   REGION External Keys /LED
       // Start Cycle
       #sStartCycle(iKeyHWStatus := "DI_PB_StartCycle",
                    oLedHWStatus => "DQ_StartCycleGreenLED");

       // Alarm Reset
       #sAlarmReset(iKeyHWStatus := "DI_PB_ResetAlarm",
                    oLedHWStatus => "DQ_AlarmBlueLED");

       // Power OFF
       #sPowerOFF(iKeyHWStatus := "DI_PB_PowerOFF",
                  oLedHWStatus => #tNoLed);

       // Shutdown PC
       #sShutdownPC(iKeyHWStatus := "DI_PB_ShutdownPC",
                    oLedHWStatus => "DQ_ShutdownPCYellowLED");

       // Light Test
       #sLightTest(iKeyHWStatus := "DI_PB_LightTest",
                   oLedHWStatus => "DQ_LightTestWhiteLED");

       // Power ON
       #sPowerON(iKeyHWStatus := "DI_PB_PowerON",
                 oLedHWStatus => "DQ_PowerOnGreenLED");

       // Remote Open Shutter
       #sRemoteOpenShutter(iKeyHWStatus := "DI_PB_RemoteOpenShutter",
                           oLedHWStatus => "DQ_RemoteOpenShutterWhiteLED");
   END_REGION

   REGION Axis Keys (Right Panel)
       #sAx10_LaserArea(iKeyHWStatus := "MCP1_In".axis10,
                        oLedHWStatus => "MCP1_Out".LEDaxis10);

       #sAx11_ChannelSelection(iKeyHWStatus := "MCP1_In".axis11,
                               oLedHWStatus => "MCP1_Out".LEDaxis11);
   END_REGION
END_FUNCTION_BLOCK

FUNCTION_BLOCK "FB_McpKeysSignals"   // FB422, SCL
{ S7_Optimized_Access := 'TRUE' }
// stored: AutoNumber false, MemoryReserve 100, SetENOAutomatically false
   VAR_INPUT
      iKeyHWStatus { ExternalAccessible := 'False'; ExternalVisible := 'False'; ExternalWritable := 'False'} : Bool;   // PLC Digital Input Hardware status
   END_VAR
   VAR_OUTPUT
      oLedHWStatus : Bool;
   END_VAR
   VAR
      sKeySWStatus : Bool;
      sKeySWToggleStatus : Bool;
      sKeyDisable : Bool;
      sKeySWPositiveFront : Bool;
      sKeySWNegativeFront : Bool;
      sKeySWTogglePositiveFront : Bool;
      sKeySWToggleNegativeFront : Bool;
      sLedSWStatus : Bool;
      sRT_KeySWPositiveFront { S7_SetPoint := 'True'} : R_TRIG;
      sFT_KeySWNegativeFront { S7_SetPoint := 'True'} : F_TRIG;
      sRT_KeySWTogglePositiveFront { S7_SetPoint := 'True'} : R_TRIG;
      sFT_KeySWToggleNegativeFront { S7_SetPoint := 'True'} : F_TRIG;
   END_VAR
BEGIN
   REGION Description header 
       //==================================================================================
       // POSALUX Swiss SA / (C) Copyright 2025
       //----------------------------------------------------------------------------------
       // Title: Management of inputs and outputs for MCP and external buttons 
       // Comment/Function: 
       //
       // Author: Fabien Waldt
       // Engineering: TIA Portal v19
       //----------------------------------------------------------------------------------
       // Change log table:
       // Version  | Date     | Expert in charge | Changes applied
       // ---------|----------|------------------|------------------------------------
       // 00.00.01 | 20250911 | WFA              | First released version
       // 00.00.02 | 20260218 | WFA              | Remove reset toggle when disable
       // ==================================================================================
   END_REGION

   REGION Inputs keys
           // Management of inputs for each customerkey MCP button 
           // Management of the software input
            IF NOT #sKeyDisable THEN
                #sKeySWStatus := #iKeyHWStatus;
            END_IF;

           // Rising/falling edge detection when pressing the button
           #sRT_KeySWPositiveFront(CLK := #sKeySWStatus,
                                  Q => #sKeySWPositiveFront);

           #sFT_KeySWNegativeFront(CLK := #sKeySWStatus,
                                  Q => #sKeySWNegativeFront);

           // Toggle state update
           IF #sKeySWPositiveFront  THEN
               #sKeySWToggleStatus := NOT #sKeySWToggleStatus;
           END_IF;

           // Rising/falling edge detection of the toggle state
           #sRT_KeySWTogglePositiveFront(CLK := #sKeySWToggleStatus,
                                        Q => #sKeySWTogglePositiveFront);

           #sFT_KeySWToggleNegativeFront(CLK := #sKeySWToggleStatus,
                                        Q => #sKeySWToggleNegativeFront);
   END_REGION

   REGION Outputs LED   
       #oLedHWStatus := #sLedSWStatus;
   END_REGION
END_FUNCTION_BLOCK

FUNCTION_BLOCK "FB_LaserAirProcess"   // FB432, SCL
{ S7_Optimized_Access := 'TRUE' }
// stored: AutoNumber false, MemoryReserve 100, SetENOAutomatically false
   VAR
      sTimeDelay : Time;
      sTimerGas : TON_TIME;
      sGasAssistOn : Bool;
      sLaser_Air_Process_Ctrl { S7_SetPoint := 'True'} : "FB_AnalogInputThreshold";
      sNozzle_Over_Pressure { S7_SetPoint := 'True'} : "FB_AnalogInputThreshold";
      sGasAssistDelay { ExternalAccessible := 'False'; ExternalVisible := 'False'; ExternalWritable := 'False'} : Bool;
      sGasAssistStartCh1 : Bool;
      sGasAssistStartCh2 : Bool;
      sGasAssistByKey : Bool;
      sGasReadValue : Bool;
      sRT_sGasAssistStartCh1 : R_TRIG;
      sRT_sGasAssistStartCh2 { S7_SetPoint := 'True'} : R_TRIG;
      sFT_sGasAssistStartCh1 { S7_SetPoint := 'True'} : F_TRIG;
      sFT_sGasAssistStartCh2 { S7_SetPoint := 'True'} : F_TRIG;
      sGasAssistSetPointJog { S7_SetPoint := 'True'} : Real;
      sGasAssistOffTimer : TOF_TIME;
   END_VAR
   VAR_TEMP
      tReadError : Bool;
      tErrorCode : Int;
   END_VAR
   VAR CONSTANT
      GAS_ASSIST_TIME : Time := T#5m;
   END_VAR
BEGIN
   REGION Description header 
       //==================================================================================
       // POSALUX Swiss SA / (C) Copyright 2024
       //----------------------------------------------------------------------------------
       // Title: Laser AirProcess
       // Comment/Function: 
       //
       // Author: Gowsigan SRITHARAN
       // Engineering: TIA Portal v17
       //----------------------------------------------------------------------------------
       // Change log table:
       // Version  | Date     | Expert in charge | Changes applied
       // ---------|----------|------------------|------------------------------------
       // 00.00.01 | 20241205 | GSR              | First released version
       // 00.00.02 | 20250314 | WFA              | Management modifications in Jog Mode
       // ==================================================================================
   END_REGION

   REGION Gas Assist ON
       "DB_DigitalOutputs".sGasAssistOn.sSWStatus := "DB_PowerOn".sMachineReadySoft;
   END_REGION

   REGION Disable Gas Assist Key[2]
       "DB_McpKeyboardSignals".sK2_GasAssist.sKeyDisable :=
       NOT "LBP_ModeGroup".E_JOG
       OR "LBP_Chan1".E_ProgRunning
       OR "LBP_Chan1".E_ProgStop
       OR "LBP_Chan1".E_ProgWait
       OR "DB_GestionWorkingModes".sMCP_KxxKeysDisable;

       "DB_HmiKeyboardSignals".sK2_GasAssist.sKeyDisable :=
       NOT "LBP_ModeGroup".E_JOG
       OR "LBP_Chan1".E_ProgRunning
       OR "LBP_Chan1".E_ProgStop
       OR "LBP_Chan1".E_ProgWait;
   END_REGION

   REGION Gas Assist
       IF "LBP_Chan1".MDyn[90] THEN                                // M90 : Start Gas Assist
           #sGasAssistStartCh1 := TRUE;
       ELSIF "LBP_Chan1".MDyn[91] OR "LBP_Chan1".A_Reset THEN      // M91 : Stop Gas Assist
           #sGasAssistStartCh1 := FALSE;
       END_IF;
   END_REGION

   REGION Gas Assist by Key
       IF "DB_McpKeyboardSignals".sK2_GasAssist.sKeySWTogglePositiveFront
           OR "DB_HmiKeyboardSignals".sK2_GasAssist.sKeySWTogglePositiveFront THEN
           #sGasAssistByKey := TRUE;
       ELSIF "DB_McpKeyboardSignals".sK2_GasAssist.sKeySWToggleNegativeFront
           OR "DB_HmiKeyboardSignals".sK2_GasAssist.sKeySWToggleNegativeFront THEN
           #sGasAssistByKey := FALSE;
       END_IF;
   END_REGION

   REGION Gas Read Value
       #sRT_sGasAssistStartCh1(CLK := #sGasAssistStartCh1);
       #sFT_sGasAssistStartCh1(CLK := #sGasAssistStartCh1);

       IF #sRT_sGasAssistStartCh1.Q
           OR #sFT_sGasAssistStartCh1.Q THEN
               #sGasReadValue := TRUE;
       END_IF;
   END_REGION

   REGION Nitrogen Gas LED[2]
       "DB_McpKeyboardSignals".sK2_GasAssist.sLedSWStatus :=
       #sGasAssistStartCh1
       OR #sGasAssistByKey;

       "DB_HmiKeyboardSignals".sK2_GasAssist.sLedSWStatus :=
       #sGasAssistStartCh1
       OR #sGasAssistByKey;
   END_REGION

   REGION Laser Air Pressure Process Set Point
       "DB_DigitalOutputs".sLaserAirPressureProcess.sSWStatus :=
       #sGasAssistStartCh1
       OR #sGasAssistByKey;
   END_REGION

   REGION Gas Assist Set point
       "LBP_TransferSelData"(Enable := #sGasReadValue,
                             Funct := 16#03,
                             IVAR1 := 972,
                             IVAR2 := -1,
                             Error => #tReadError,
                             ErrCode => #tErrorCode,
                             S7Var := "DB_HMISetting".GasAssistSetPoint);

       // Gas Assist Set Point if Jog mode
       IF NOT "LBP_ModeGroup".E_JOG AND "DB_HMISetting".GasAssistSetPoint <> 0 AND #sGasReadValue THEN
           #sGasAssistSetPointJog := "DB_HMISetting".GasAssistSetPoint;
       ELSE
           #sGasAssistSetPointJog := "DB_Parameters".GazPressureManual;
        END_IF;   

       // Transfer Gas Assist Set Point
        IF #sGasReadValue THEN
           IF "LBP_ModeGroup".E_JOG THEN
               "DB_AnalogInputDataHMI".Laser_Air_Pressure_Process.TargetValue := #sGasAssistSetPointJog;
               "DB_AnalogInputDataHMI".Nozzle_Overpressure.TargetValue := #sGasAssistSetPointJog;
           ELSE
               "DB_AnalogInputDataHMI".Laser_Air_Pressure_Process.TargetValue := "DB_HMISetting".GasAssistSetPoint;
               "DB_AnalogInputDataHMI".Nozzle_Overpressure.TargetValue := "DB_HMISetting".GasAssistSetPoint;
           END_IF;
       END_IF;

       // Reset Gas Assist Value by push Reset Button or after 5min no process
       #sGasAssistOffTimer(IN := ("LBP_Chan1".E_ProgRunning AND "LBP_Chan1".E_ProgRunning)
                           OR ("LBP_ModeGroup".E_JOG AND "DB_McpKeyboardSignals".sK2_GasAssist.sKeySWToggleStatus)
                           OR ("LBP_ModeGroup".E_JOG AND "DB_HmiKeyboardSignals".sK2_GasAssist.sKeySWToggleStatus),
                           PT := #GAS_ASSIST_TIME);

       // IF "MCP1_In".reset OR NOT #sGasAssistOffTimer.Q THEN
           IF "MCP1_In".reset THEN // WFA A REVOIR
           "DB_HMISetting".GasAssistSetPoint := 0.0;
           "DB_AnalogInputDataHMI".Laser_Air_Pressure_Process.TargetValue := 0.0;
           "DB_AnalogInputDataHMI".Nozzle_Overpressure.TargetValue := 0.0;
       END_IF;

       // Gas assist transfer to analog output
       IF NOT "LBP_ModeGroup".E_JOG THEN
           "DB_AnalogOutputs".sNozzleOverpressureSetPoint.sSWRealValue := "DB_HMISetting".GasAssistSetPoint;
       ELSE
           "DB_AnalogOutputs".sNozzleOverpressureSetPoint.sSWRealValue := #sGasAssistSetPointJog;
       END_IF;
   END_REGION

   REGION Laser Air process control
       #sLaser_Air_Process_Ctrl(iActualValue := "DB_AnalogInputs".sLaserAirPressureProcess.sSWRealValue,
                                iStartDelay := "DB_DigitalOutputs".sLaserAirPressureProcess.sSWStatus,
                                ioAlarmMin := "LBP_AlarmMsgs".UserA[06].A70UUxx[50],
                                ioWarningMin := "LBP_AlarmMsgs".UserA[07].A70UUxx[50],
                                ioWarningMax := "LBP_AlarmMsgs".UserA[07].A70UUxx[51],
                                ioAlarmMax := "LBP_AlarmMsgs".UserA[06].A70UUxx[51],
                                oDataAction => "DB_AnalogInputAction".Laser_Air_Pressure_Process,
                                iDataPLC := "DB_AnalogInputDataPLC".Laser_Air_Pressure_Process,
                                iDataHMI := "DB_AnalogInputDataHMI".Laser_Air_Pressure_Process);
     END_REGION

     REGION Regulation gas assist control
         #sNozzle_Over_Pressure(iActualValue := "DB_AnalogInputs".sNozzleOverpressure.sSWRealValue,
                                iStartDelay := "DB_DigitalOutputs".sLaserAirPressureProcess.sSWStatus,
                                ioAlarmMin := "LBP_AlarmMsgs".UserA[06].A70UUxx[60],
                                ioWarningMin := "LBP_AlarmMsgs".UserA[07].A70UUxx[60],
                                ioWarningMax := "LBP_AlarmMsgs".UserA[07].A70UUxx[61],
                                ioAlarmMax := "LBP_AlarmMsgs".UserA[06].A70UUxx[61],
                                oDataAction => "DB_AnalogInputAction".Nozzle_Overpressure,
                                iDataPLC := "DB_AnalogInputDataPLC".Nozzle_Overpressure,
                                iDataHMI := "DB_AnalogInputDataHMI".Nozzle_Overpressure);
     END_REGION
END_FUNCTION_BLOCK

FUNCTION_BLOCK "FB_AnalogInputThreshold"   // FB221, SCL
{ S7_Optimized_Access := 'TRUE' }
// stored: AutoNumber false, MemoryReserve 100, SetENOAutomatically false
   VAR_INPUT
      iActualValue : Real;
      iStartDelay : Bool;
      iDataPLC { ExternalAccessible := 'False'; ExternalVisible := 'False'; ExternalWritable := 'False'} : "AnalogInDataPLC_DT";
      iDataHMI { ExternalAccessible := 'False'; ExternalVisible := 'False'; ExternalWritable := 'False'} : "AnalogInDataHMI_DT";
   END_VAR
   VAR_OUTPUT
      oDataAction { ExternalAccessible := 'False'; ExternalVisible := 'False'; ExternalWritable := 'False'} : "AnalogInAction_DT";
   END_VAR
   VAR_IN_OUT
      ioAlarmMin : Bool;
      ioWarningMin : Bool;
      ioWarningMax : Bool;
      ioAlarmMax : Bool;
   END_VAR
   VAR
      sStartTimer : TON_TIME;
      sTONAlarmMin : TON_TIME;
      sTONWarningMin : TON_TIME;
      sTONWarningMax : TON_TIME;
      sTONAlarmMax : TON_TIME;
      sMemoAlarmMin { S7_SetPoint := 'True'} : Bool;
      sMemoWarningMin { S7_SetPoint := 'True'} : Bool;
      sMemoWarningMax { S7_SetPoint := 'True'} : Bool;
      sMemoAlarmMax { S7_SetPoint := 'True'} : Bool;
   END_VAR
BEGIN
   REGION Description header 
       //==================================================================================
       // POSALUX Swiss SA / (C) Copyright 2024
       //----------------------------------------------------------------------------------
       // Title: Analog input management 
       // Comment/Function: This function manages alarms and warnings based on a  
       //                   current value compared to predefined target. After an
       //                   initial delay, it activates specific alarms OR warnings if the
       //                   value exceeds thresholds, and can also trigger machine
       //                   shutdown or signal a defective part according TO conditions
       //                   configured on the HMI.
       // Author: Gowsigan SRITHARAN
       // Engineering: TIA Portal v17
       //----------------------------------------------------------------------------------
       // Change log table:
       // Version  | Date     | Expert in charge | Changes applied
       // ---------|----------|------------------|------------------------------------
       // 00.00.01 | 20241121 | GSR              | First released version
       // 00.00.02 | 20250911 | WFA              | Work with target
       // ==================================================================================
   END_REGION

   REGION Start Timer
       #sStartTimer(IN := #iStartDelay,
                    PT := #iDataHMI.StartTime);
       #sTONAlarmMin(IN := #sMemoAlarmMin,
                     PT := #iDataPLC.DelayAlarmMin);
       #sTONWarningMin(IN := #sMemoWarningMin,
                       PT := #iDataPLC.DelayWarningMin);
       #sTONAlarmMax(IN := #sMemoAlarmMax,
                     PT := #iDataPLC.DelayAlarmMax);
       #sTONWarningMax(IN := #sMemoWarningMax,
                       PT := #iDataPLC.DelayWarningMax);
   END_REGION

   REGION Detect alarm/warning
       IF #sStartTimer.Q THEN
           #sMemoWarningMin := #iDataHMI.TargetValue + #iDataHMI.ThresholdWarningMin >= #iActualValue AND #iDataPLC.EnableWarningMin AND NOT #sMemoAlarmMin;

           #sMemoWarningMax := #iDataHMI.TargetValue + #iDataHMI.ThresholdWarningMax <= #iActualValue AND #iDataPLC.EnableWarningMax AND NOT #sMemoAlarmMax;

           #sMemoAlarmMin := #iDataHMI.TargetValue + #iDataHMI.ThresholdAlarmMin >= #iActualValue AND #iDataPLC.EnableAlarmMin;

           #sMemoAlarmMax := #iDataHMI.TargetValue + #iDataHMI.ThresholdAlarmMax <= #iActualValue AND #iDataPLC.EnableAlarmMax;
       ELSE
           #sMemoWarningMin := FALSE;
           #sMemoWarningMax := FALSE;
           #sMemoAlarmMin   := FALSE;
           #sMemoAlarmMax   := FALSE;
       END_IF;

   END_REGION

   REGION Set alarm/warning
       // Alarme Min
       IF #sTONAlarmMin.Q THEN
           #ioAlarmMin := TRUE;
           #ioWarningMin := FALSE;
           #oDataAction.BadPartOnFixture := #iDataPLC.BadPartOnFixture; // Set bad part if alarm
           #oDataAction.ID_Measure := #iDataHMI.ID_Measure;
       ELSE
           #oDataAction.BadPartOnFixture := FALSE;
           #oDataAction.ID_Measure := 0;
       END_IF;

       // Warning Min
       IF #sTONWarningMin.Q THEN
           #ioWarningMin := TRUE;
       END_IF;

       // Alarm Max
       IF #sTONAlarmMax.Q THEN
           #ioAlarmMax := TRUE;
           #ioWarningMax := FALSE;
           #oDataAction.BadPartOnFixture := #iDataPLC.BadPartOnFixture; // Set bad part if alarm
           #oDataAction.ID_Measure := #iDataHMI.ID_Measure;
       ELSE
           #oDataAction.BadPartOnFixture := FALSE;
           #oDataAction.ID_Measure := 0;
       END_IF;

       // Warning Max
       IF #sTONWarningMax.Q THEN
           #ioWarningMax := TRUE;
       END_IF;
   END_REGION
END_FUNCTION_BLOCK

FUNCTION_BLOCK "FB_LaserOperation"   // FB431, SCL
{ S7_Optimized_Access := 'TRUE' }
// stored: AutoNumber false, MemoryReserve 100, SetENOAutomatically false
   VAR
      sLaserTimeCh1 : "FB_TimeCounter";
      sLaserCycleTimeCh1 { S7_SetPoint := 'True'} : Int;
   END_VAR
BEGIN
   REGION Description header 
       //==================================================================================
       // POSALUX Swiss SA / (C) Copyright 2024
       //----------------------------------------------------------------------------------
       // Title: Laser AirProcess
       // Comment/Function: 
       //
       // Author: Gowsigan SRITHARAN
       // Engineering: TIA Portal v17
       //----------------------------------------------------------------------------------
       // Change log table:
       // Version  | Date     | Expert in charge | Changes applied
       // ---------|----------|------------------|------------------------------------
       // 00.00.01 | 20241205 | GSR              | First released version
       // ==================================================================================
   END_REGION

   REGION Head Laser Circuit breaker
       IF NOT "DB_DigitalInputs".sHeadLaserBreaker.sSWStatus THEN
           "LBP_AlarmMsgs".UserA[0].A70UUxx[2] := TRUE;
       END_IF;
   END_REGION

   REGION Head_Laser start and stop
       "DB_DigitalOutputs".sHeadLaserStart.sSWStatus := "DB_PowerOn".sMachineReadySoft;
       "DB_DigitalOutputs".sHeadLaserStop.sSWStatus  := "DB_PowerOn".sMachineReadySoft;
   END_REGION

   REGION LED laser button 
       IF ("DB_DataFromSafety".ShutterOpened
           AND NOT "DB_DataFromSafety".ShutterClosed)
           OR "DB_McpKeyboardSignals".sLightTest.sKeySWStatus THEN  // Test Lamp
           "DB_McpKeyboardSignals".sRemoteOpenShutter.sLedSWStatus := TRUE;
       ELSIF "DB_DataFromSafety".ShutterClosed AND NOT "DB_DataFromSafety".ShutterOpened THEN
           IF "DB_DataFromSafety".ShutterReadyToOpen THEN
               // Ready to open -> slow blinking
               "DB_McpKeyboardSignals".sRemoteOpenShutter.sLedSWStatus := "Clock_0.5Hz";
           ELSIF "DB_DataFromSafety".OpenShutter THEN
               // Ready to open -> quick blinking
               "DB_McpKeyboardSignals".sRemoteOpenShutter.sLedSWStatus := "Clock_2Hz";
           ELSE
               // Close -> off
               "DB_McpKeyboardSignals".sRemoteOpenShutter.sLedSWStatus := FALSE;
           END_IF;
       ELSE
           // Close -> off
           "DB_McpKeyboardSignals".sRemoteOpenShutter.sLedSWStatus := FALSE;
       END_IF;
   END_REGION

   REGION Laser Key ON / Shutter closed
       "DB_HMIStatus".KeyLaserOn := "DB_DataFromSafety".iKeyLaserOn;
       "DB_HMIStatus".Shutter_laser_closed := "DB_DigitalInputs".sShutterClosed.sSWStatus OR NOT "DB_DataFromSafety".iKeyLaserOn;
   END_REGION


   REGION Laser Cycle Time
       #sLaserTimeCh1(iStart := "LBP_Chan1".MDyn[71],                        // M71 : Start calculation laser time 
                      iReset := "LBP_Chan1".MDyn[68] OR "MCP1_In".reset);    // M68 : Reset calculation laser time 
       #sLaserCycleTimeCh1 := #sLaserTimeCh1.ioMinutesCumul;
   END_REGION
END_FUNCTION_BLOCK

FUNCTION_BLOCK "FB_TimeCounter"   // FB53, SCL
{ S7_Optimized_Access := 'TRUE' }
// stored: MemoryReserve 100, SetENOAutomatically false
   VAR_INPUT
      iStart : Bool;
      iReset : Bool;
   END_VAR
   VAR_IN_OUT
      ioHours : Int;
      ioMinutes : Int;
      ioSeconds : Int;
      ioHoursCumul : Int;
      ioMinutesCumul : Int;
      ioSecondsCumul : DInt;
   END_VAR
   VAR
      sRT_Second { ExternalAccessible := 'False'; ExternalVisible := 'False'; ExternalWritable := 'False'} : R_TRIG;
   END_VAR
BEGIN
   REGION Description header 
       //==================================================================================
       // POSALUX Swiss SA / (C) Copyright 2025
       //----------------------------------------------------------------------------------
       // Title: Timer Counter
       // Comment/Function: This function allows:
       //                      - Counting Hours - Minutes - Seconds 
       //                      - Pulse each Hour - Minute - Second
       //
       // Author: Fabien Waldt
       // Engineering: TIA Portal v17
       //----------------------------------------------------------------------------------
       // Change log table:
       // Version  | Date     | Expert in charge | Changes applied
       // ---------|----------|------------------|------------------------------------
       // 00.00.01 | 20250314 | WFA              | First released version
       // ==================================================================================
   END_REGION

   //"Seconds" rising edge
   #sRT_Second(CLK := "Clock_1Hz");

   REGION Time counters reset
       IF #iReset THEN
           #ioHours := 0;
           #ioMinutes := 0;
           #ioSeconds := 0;
           #ioHoursCumul := 0;
           #ioMinutesCumul := 0;
           #ioSecondsCumul := 0;
       END_IF;
   END_REGION

   REGION Time counters
   IF #iStart AND #sRT_Second.Q THEN
       #ioSeconds := #ioSeconds + 1;
       #ioSecondsCumul := #ioSecondsCumul + 1;
       IF #ioSeconds >= 60 THEN
           #ioMinutes := #ioMinutes + 1;
           #ioSeconds := 0;
           #ioMinutesCumul := #ioMinutesCumul + 1;
           IF #ioMinutes >= 60 THEN
               #ioHours := #ioHours + 1;
               #ioMinutes := 0;
               #ioHoursCumul := #ioHoursCumul + 1;
           END_IF;
       END_IF;
   END_IF;
   END_REGION
END_FUNCTION_BLOCK

FUNCTION_BLOCK "FB_LaserMeasureZoneSwitch"   // FB417, SCL
{ S7_Optimized_Access := 'TRUE' }
// stored: AutoNumber false, MemoryReserve 100, SetENOAutomatically false
   VAR RETAIN
      sMeasure1 : Bool;   // Limit sw Measure 1 / Axes are on Area Measure station 1
      sMeasure2 : Bool;   // Limit sw Measure 2 / Axes are on Area Measure station 2
      sLaser1 : Bool;   // Condition Laser 1 / Gate for going to area laser Station 1
      sLaser2 : Bool;   // Condition Laser 2 / Gate for going to area laser Station 2
      sLaserArea1Req : Bool;   // Laser area 1 request / Ask for going to laser Area Station 1
      sLaserArea2Req : Bool;   // Laser area 2 request / Ask for going to laser Area Station 2
      sCuttingArea1Req : Bool;   // Cutting 1 request / Axe X1 enter to laser Area
      sCuttingArea2Req : Bool;   // Cutting 2 request / Axe X2 enter to laser Area
      sCutBusy : Bool;   // ???
      sCut1 : Bool;   // Axe X1 traverse the gate (X1SoftLimMin1)
      sCut2 : Bool;   // Axe X2 traverse the gate (X1SoftLimMin1)
      sX1Pos : Real;
      sX2Pos : Real;
   END_VAR
   VAR
      sRT_GateCut1 : R_TRIG;
      sRT_GateCut2 : R_TRIG;
   END_VAR
   VAR RETAIN
      sCondDegageAxe : Bool;
      sRefAxisActive : Bool;
   END_VAR
BEGIN
   REGION Description header 
       //==================================================================================
       // POSALUX Swiss SA / (C) Copyright 2025
       //----------------------------------------------------------------------------------
       // Title: FB_ManageLaserOrMeasureArea
       // Comment/Function: manages two zones (laser or measurement) on two statio
       // ns, if
       // present, based on the position of the axes and/or the state of a keyboard button.
       //It dynamically switches the software limits OF the axes (limit 1 OR 2) according
       //TO the active zone, allowing the machine’s safety AND behavior TO adapt TO each
       //operating mode.
       // Author: Fabien Waldt
       // Engineering: TIA Portal v17
       //----------------------------------------------------------------------------------
       // Change log table:
       // Version  | Date     | Expert in charge | Changes applied
       // ---------|----------|------------------|------------------------------------
       // 00.00.01 | 20250224 | FWA              | First released version
       // ==================================================================================
   END_REGION

   REGION Key [16] Disable + Toggle
       // Disable Key [16] - collision detection of the ZL axis with the X axis // WFA ??
       "DB_McpKeyboardSignals".sAx10_LaserArea.sKeyDisable := NOT "LBP_ModeGroup".E_JOG;
       //On channel change, update the MCP button to reflect the toggle status of the newly selected channel 
       // "DB_McpKeyboardSignals".Ax10_LaserArea.KeySWToggleStatus :=
       // (#LaserArea1Req AND "DB_DecodChannels".Chan1IsDisplayed);
   END_REGION

   REGION Laser Area 1 Request
       IF "LBP_Chan1".MDyn[60]     // M60: Axes Limit for Laser Area
           OR ("DB_McpKeyboardSignals".sAx10_LaserArea.sKeySWTogglePositiveFront  AND "DB_DecodChannels".sChan1IsDisplayed) THEN
           #sLaserArea1Req := TRUE;
           "LBP_AlarmMsgs".ChanA[1].RID_5C02xx[0] := TRUE;         // Msg: "510200 - Waiting gate laser - M60"
       END_IF;

       IF "LBP_Chan1".MDyn[61]     // M61: Axes Limit for Measure Area
           OR ("DB_McpKeyboardSignals".sAx10_LaserArea.sKeySWToggleNegativeFront AND "DB_DecodChannels".sChan1IsDisplayed) THEN
           #sLaserArea1Req := FALSE;
           "LBP_AlarmMsgs".ChanA[1].RID_5C02xx[1] := TRUE;    // Msg: "510201 - Waiting gate measure - M61"
       END_IF;


   END_REGION

   REGION Conditions to switch the limit of axis
       IF #sLaserArea1Req 
           AND ("DB_AxisPosition".sAxis03_ZM."$AA_IM" >= "DB_AxisPosition".sAxis03_ZM."$MA_POS_LIMIT_MINUS2")  // ZM upper as limit M2
           AND ("DB_AxisPosition".sAxis04_B."$AA_IM" >= "DB_AxisPosition".sAxis04_B."$MA_POS_LIMIT_MINUS2")    // B upper as limit M2
           AND ("DB_AxisPosition".sAxis07_V."$AA_IM" <= "DB_AxisPosition".sAxis07_V."$MA_POS_LIMIT_PLUS2")     // V below as limit P2
           AND ("DB_AxisPosition".sAxis02_Y."$AA_IM" <= "DB_AxisPosition".sAxis02_Y."$MA_POS_LIMIT_PLUS2")     // Y below as limit P2
           AND "DB_Powermeter".sPowermeterInHomePos THEN   // Powermeter retracted
               #sLaser1 := TRUE;    // Set Laser 1
               #sMeasure1 := FALSE;
      ELSIF NOT #sLaserArea1Req AND
          ("DB_AxisPosition".sAxis01_X."$AA_IM" <= "DB_AxisPosition".sAxis01_X."$MA_POS_LIMIT_PLUS") THEN   // X below as limit P1
               #sMeasure1 := TRUE;
               #sLaser1 := FALSE;
       ELSE
           #sMeasure1 := FALSE;
       END_IF;
   END_REGION

   REGION Switch of the limit of axis (laser --> limit 2 / Measure --> Limit 1)
       IF #sLaser1 THEN
           "LBP_Axis01_X".A_SWLimit2Plus := TRUE;
           "LBP_Axis02_Y".A_SWLimit2Plus := TRUE;
           "LBP_Axis03_ZM".A_SWLimit2Plus := TRUE;
           "LBP_Axis04_B".A_SWLimit2Plus := TRUE;
           "LBP_Axis07_V".A_SWLimit2Plus := TRUE;
       ELSIF #sMeasure1 THEN
           "LBP_Axis01_X".A_SWLimit2Plus := FALSE;
           "LBP_Axis02_Y".A_SWLimit2Plus := FALSE;
           "LBP_Axis03_ZM".A_SWLimit2Plus := FALSE;
           "LBP_Axis04_B".A_SWLimit2Plus := FALSE;
           "LBP_Axis07_V".A_SWLimit2Plus := FALSE;
       END_IF;
   END_REGION

   REGION Led of the MCP button

       "DB_McpKeyboardSignals".sAx10_LaserArea.sLedSWStatus :=
       ((#sLaserArea1Req AND #sLaser1)
       OR (#sLaserArea1Req AND NOT #sLaser1 AND "Clock_1Hz")
       OR (NOT #sLaserArea1Req AND NOT #sLaser1 AND "Clock_1Hz"))
       AND "DB_DecodChannels".sChan1IsDisplayed
       OR ((#sLaserArea2Req AND #sLaser2)
       OR (#sLaserArea2Req AND NOT #sLaser2 AND "Clock_1Hz")
       OR (NOT #sLaserArea2Req AND NOT #sLaser2 AND "Clock_1Hz"))
       AND "DB_DecodChannels".sChan2IsDisplayed;
   END_REGION

   REGION Read in disable
       // Read in disable: laser 1 : gate NOT ready
       IF NOT #sLaserArea1Req OR #sLaser1 OR "LBP_Chan1".A_Reset THEN
           "LBP_AlarmMsgs".ChanA[1].RID_5C02xx[0] := FALSE;
       END_IF;
       IF #sLaserArea1Req OR #sMeasure1 OR "LBP_Chan1".A_Reset THEN
           "LBP_AlarmMsgs".ChanA[1].RID_5C02xx[1] := FALSE;
       END_IF;
   END_REGION

   REGION Anticollision - A REVOIR LORS MISE EN ROUTE
       REGION Conditions de dégagement
           #sCondDegageAxe := "LBP_ModeGroup".E_JOG AND NOT "LBP_ModeGroup".E_REF;
       END_REGION

       REGION Machine en Ref Active
           #sRefAxisActive := "LBP_Chan1".A_Ref OR "LBP_Chan2".A_Ref;
       END_REGION

       REGION Anticollision entre X1/V1
           IF "LBP_Axis01_X".A_SWLimit2Minus// Ne sert plus a rien car 0<v<200 
               AND ("DB_AxisPosition".sAxis07_V."$AA_IM" >= 9999.9999) THEN
               "LBP_AlarmMsgs".Axis[01].FdStop[10] := TRUE;
               "LBP_AlarmMsgs".Axis[07].FdStop[10] := TRUE;
            //   "LBP_AlarmMsgs".UserA[2].A70UUxx[10] := TRUE;   // Msg: "702010 - ???"
           END_IF;
           //Pas compris pour eviter collision avec x1 et v1
           IF (#sCondDegageAxe AND "LBP_Axis07_V".E_TCMinus)
               OR NOT "DB_DataToSafety".FrontDoorLock
               OR #sRefAxisActive THEN
               "LBP_AlarmMsgs".Axis[01].FdStop[10] := FALSE;
               "LBP_AlarmMsgs".Axis[07].FdStop[10] := FALSE;
            //   "LBP_AlarmMsgs".UserA[2].A70UUxx[10] := FALSE;   // Msg: "702010 - ???"
           END_IF;
       END_REGION

       REGION Anticollision entre X1/ZM1
           IF "LBP_Axis01_X".A_SWLimit2Minus // Ne sert plus a rien car -22<ZM1<160 
               AND (9999.9999 <= "DB_AxisPosition".sAxis03_ZM."$AA_IM") THEN
               "LBP_AlarmMsgs".Axis[01].FdStop[10] := TRUE;
               "LBP_AlarmMsgs".Axis[03].FdStop[10] := TRUE;
            //   "LBP_AlarmMsgs".UserA[2].A70UUxx[11] := TRUE;   // Msg: "702011 - ???"
           END_IF;
           //Pas compris pour eviter collision avec x1 et v1
           IF (#sCondDegageAxe AND "LBP_Axis03_ZM".E_TCPlus)
               OR NOT "DB_DataToSafety".FrontDoorLock
               OR #sRefAxisActive THEN
               "LBP_AlarmMsgs".Axis[01].FdStop[10] := FALSE;
               "LBP_AlarmMsgs".Axis[03].FdStop[10] := FALSE;
          //   "LBP_AlarmMsgs".UserA[2].A70UUxx[11] := FALSE;   // Msg: "702011 - ???"
           END_IF;
       END_REGION
   END_REGION

   REGION Cutting
       // WFA VOIR SI CUTTING NECESSAIRE POUR MACHINE MONO
       REGION Cutting : M62 waiting laser cutting free
           IF "LBP_Chan1".MDyn[62] THEN    // M62: Axes Limit for Cutting Area
               #sCuttingArea1Req := TRUE;
               "LBP_AlarmMsgs".ChanA[1].RID_5C02xx[2] := TRUE;         // Msg: "510202 - Waiting laser"
               #sX1Pos := LREAL_TO_REAL("DB_AxisPosition".sAxis01_X."$AA_IM");
           END_IF;
       END_REGION

       REGION Set cutting busy by X pos : JOG, man, prog interrupt, prog err
           #sRT_GateCut1(CLK := "DB_AxisPosition".sAxis01_X."$AA_IM" < "DB_AxisPosition".sAxis01_X."$A1_M_FP_POS4_30600");
           IF #sRT_GateCut1.Q THEN
               #sCut1 := TRUE;
           END_IF;
       END_REGION

       REGION X collision avoid
           IF #sCut1 AND #sCut2 THEN
               "LBP_AlarmMsgs".Axis[1].FdStop[0] := TRUE;
               "LBP_AlarmMsgs".Axis[10].FdStop[0] := TRUE;
           END_IF;

           // X1 plus: R stop X1
           IF "LBP_Chan1".E_ChanReset
               OR "LBP_Axis01_X".E_TCPlus
               OR "LBP_Chan1".A_Reset
               OR ("LBP_ModeGroup".E_JOG AND "LBP_ModeGroup".E_REF) THEN
               "LBP_AlarmMsgs".Axis[1].FdStop[0] := FALSE;
           END_IF;
           //check programmed X destination position
           //if in cuting area without gate_cut:stop
       END_REGION

       REGION Open cutting laser gate
           IF #sCuttingArea1Req THEN
               #sCut1 := TRUE;
               // ZL Get -> chan 1
               "LBP_Axis09_ZL".A_NCASpStrobe := TRUE;
               "LBP_Axis09_ZL".A_NCASpChanB := FALSE;
               "LBP_Axis09_ZL".A_NCASpChanA := TRUE;
           END_IF;
       END_REGION
       REGION Reset Gate_Cut_1 and Gate_Cut_2
           IF #sX1Pos >= "DB_AxisPosition".sAxis01_X."$A1_M_FP_POS4_30600" THEN
               #sX1Pos := LREAL_TO_REAL("DB_AxisPosition".sAxis01_X."$A1_M_FP_POS4_30600");
           END_IF;

           IF #sX1Pos + 1.0 < "DB_AxisPosition".sAxis01_X."$AA_IM" OR
               "LBP_Chan1".MDyn[63] THEN
               #sCut1 := FALSE;
           END_IF;
       END_REGION

       REGION Release M62
           // IF #sCut1 AND
           //     "LBP_Axis09_ZL".E_NCASpChanA
           //     AND NOT "LBP_Axis09_ZL".E_NCASpChanB
           //     OR "LBP_Chan1".A_Reset THEN
           //     "LBP_Axis09_ZL".A_NCASpStrobe := FALSE;
           //     #sCuttingArea1Req := FALSE;
           IF "DB_OPC_Laser".Scanner.In.Ready THEN
               "LBP_AlarmMsgs".ChanA[1].RID_5C02xx[2] := FALSE;         // Msg: "510202 - Waiting laser"
           END_IF;
       END_REGION
   END_REGION
   //Copie de la FL0125, Pas sur que ca existe sur les FEMTO 5A mono ou twin
   //A voir egalement les colisions à partir du code de la FL0107

   // REGION NETWORK 34
   //     IF "LBP_Chan1".MDyn[62] THEN    // M62: Axes Limit for Cutting Area
   //         #CuttingArea1Req := TRUE;
   //         "LBP_AlarmMsgs".ChanA[1].RID_5C02xx[2] := TRUE;
   //         #X1_POS := LREAL_TO_REAL("DB_AxisPosition_ReadVar".sAxis01_X1."$AA_IM");
   //     END_IF;

   //     IF "LBP_Chan2".MDyn[62] THEN    // M62: Axes Limit for Cutting Area
   //         #CuttingArea2Req := TRUE;
   //         "LBP_AlarmMsgs".ChanA[2].RID_5C02xx[2] := TRUE;
   //         #X2_POS := LREAL_TO_REAL("DB_AxisPosition_ReadVar".sAxis10_X2."$AA_IM");
   //     END_IF;
   // END_REGION

   // REGION NETWORK 35
   //     // WFA A REVOIR
   //     #Gate_Cut_1 := FALSE;
   //     #Gate_Cut_2 := FALSE;
   // END_REGION

   // REGION NETWORK 36
   //     IF #Gate_Cut_1 AND #Gate_Cut_2 THEN
   //         "LBP_AlarmMsgs".Axis[1].FdStop[0] := TRUE;
   //         "LBP_AlarmMsgs".Axis[10].FdStop[0] := TRUE;
   //     END_IF;

   //     //x1 plus: R stop x1
   //     IF "LBP_Chan1".E_ChanReset
   //         OR "LBP_Axis01_X1".E_TCPlus
   //         OR "LBP_Chan1".A_Reset
   //         OR ("LBP_ModeGroup".E_JOG AND "LBP_ModeGroup".E_REF) THEN
   //         "LBP_AlarmMsgs".Axis[1].FdStop[0] := FALSE;
   //     END_IF;

   //     //x2 minus: R stop x2
   //     IF "LBP_Chan2".E_ChanReset
   //         OR "LBP_Axis10_X2".E_TCMinus
   //         OR "LBP_Chan2".A_Reset
   //         OR ("LBP_ModeGroup".E_JOG AND "LBP_ModeGroup".E_REF) THEN
   //         "LBP_AlarmMsgs".Axis[10].FdStop[0] := FALSE;
   //     END_IF;


   //     //check programmed X destination position
   //     //if in cuting area without gate_cut:stop
   // END_REGION

   // REGION NETWORK 37
   //     IF #CuttingArea1Req AND NOT #Gate_Cut_2 THEN
   //         #Gate_Cut_1 := TRUE;
   //         "LBP_Axis09_ZL".A_NCASpStrobe := TRUE;
   //         "LBP_Axis09_ZL".A_NCASpChanB := FALSE;
   //         "LBP_Axis09_ZL".A_NCASpChanA := TRUE;
   //     END_IF;

   //     IF #CuttingArea2Req AND NOT #Gate_Cut_2 THEN
   //         #Gate_Cut_2 := TRUE;
   //         "LBP_Axis09_ZL".A_NCASpStrobe := TRUE;
   //         "LBP_Axis09_ZL".A_NCASpChanB := TRUE;
   //         "LBP_Axis09_ZL".A_NCASpChanA := FALSE;
   //     END_IF;
   // END_REGION

   // REGION NETWORK 38
   //     // WFA A REVOIR
   //     IF #X1_POS + 1.0 < "DB_AxisPosition_ReadVar".sAxis01_X1."$AA_IM" OR
   //         "LBP_Chan1".MDyn[63] THEN
   //         #Gate_Cut_1 := FALSE;
   //     END_IF;

   //     IF #X2_POS + 1.0 < "DB_AxisPosition_ReadVar".sAxis10_X2."$AA_IM" OR
   //         "LBP_Chan2".MDyn[63] THEN
   //         #Gate_Cut_2 := FALSE;
   //     END_IF;
   // END_REGION


   // REGION NETWORK 39
   //     IF #Gate_Cut_1 AND
   //         "LBP_Axis09_ZL".E_NCASpChanA
   //         AND NOT "LBP_Axis09_ZL".E_NCASpChanB
   //         OR "LBP_Chan1".A_Reset THEN
   //         "LBP_Axis09_ZL".A_NCASpStrobe := FALSE;
   //         #CuttingArea1Req := FALSE;
   //         "LBP_AlarmMsgs".ChanA[1].RID_5C02xx[2] := FALSE;
   //     END_IF;

   //     IF #Gate_Cut_2 AND
   //         NOT "LBP_Axis09_ZL".E_NCASpChanA
   //         AND "LBP_Axis09_ZL".E_NCASpChanB
   //         OR "LBP_Chan2".A_Reset THEN
   //         "LBP_Axis09_ZL".A_NCASpStrobe := FALSE;
   //         #CuttingArea2Req := FALSE;
   //         "LBP_AlarmMsgs".ChanA[2].RID_5C02xx[2] := FALSE;
   //     END_IF;
   // END_REGION
END_FUNCTION_BLOCK

FUNCTION_BLOCK "FB_Powermeter"   // FB433, SCL
{ S7_Optimized_Access := 'TRUE' }
// stored: AutoNumber false, MemoryReserve 100, SetENOAutomatically false
   VAR
      sPowerMeterWorkPos : Bool;
      sPowerMeterHomePos : Bool;
      sPowerMeterToWorkMoveReq : Bool;
      sPowerMeterToHomeMoveReq : Bool;
      sPowerMeterJogMode : Bool;
      sPowermeterCylinder : "FB_CmdCylinder";
      sPowermeterInHomePos { S7_SetPoint := 'True'} : Bool;
      sPowermeterInMiddlePos : Bool;
      sPowermeterInWorkPos : Bool;
      sPowerMeterCylErrorCode : Int;
      sPowerMeterHomePosCtrlTimer : TON_TIME;
      sPowerMeterWorkPosCtrlTimer : TON_TIME;
      sMeasurePowerLaser { S7_SetPoint := 'True'} : Bool;
      sRTLaserMeasureON : R_TRIG;
      sLaserPowerValue { S7_SetPoint := 'True'} : Real;
      sWeightFactor : Real;
      sAlpha : Real;
      sDateAndTime : DTL;
      sActualMeasPower : Real;
      sTolMin : Real;
      sTolMax : Real;
      sResetMeasures : Bool;
      sPowerMeterSeq : "FB_PowerMeterSeq";
      RT_StartArchive { S7_SetPoint := 'True'} : R_TRIG;
      sArchivePmValues { S7_SetPoint := 'True'} : Array[0..4] of Real;
   END_VAR
   VAR_TEMP
      tAxis01_X1SafePos : Bool;
      tLaserMeasureON : Bool;
      tActualMeasure : Int;
      tRetVal : Int;
      tAverageValue : Real;
      tStandardDeviation : Real;
      tTempReal : Real;
      tIndex : Int;
   END_VAR
   VAR CONSTANT
      POWERMETER_HOME_POS_CTRL_TIME : Time := T#6s;
      POWERMETER_WORK_POS_CTRL_TIME : Time := T#6s;
   END_VAR
BEGIN
   REGION Description header 
       //==================================================================================
       // POSALUX Swiss SA / (C) Copyright 2025
       //----------------------------------------------------------------------------------
       // Title: Initialization of axis
       // Comment/Function: 
       // Author: Fabien WALDT
       // Engineering: TIA Portal v17
       //----------------------------------------------------------------------------------
       // Change log table:
       // Version  | Date     | Expert in charge | Changes applied
       // ---------|----------|------------------|-----------------------------------------
       // 00.00.01 | 20250501 | WFA              | First released version
       // =================================================================================
   END_REGION

   REGION Axis01_X on safe position
      // Check position Axis01_X to release the powermeter
       #tAxis01_X1SafePos := "DB_AxisPosition".sAxis01_X."$AA_IM" >= "DB_AxisPosition".sAxis01_X."$MA_POS_LIMIT_PLUS" - 10.0;
   END_REGION

   REGION Blocking Axis01_X
       // Blocking Axis01_X if Powermeter is in measuring position
       "LBP_Axis01_X".A_ASpDisable := NOT #sPowerMeterHomePos OR #sPowerMeterWorkPos; 
   END_REGION
   REGION PowerMeter Sequence
       // #sPowerMeterSeq(iStartSeqCond:=#sPowerMeterSeq.iStartSeqCond,
       //                 iJobReq:=#sPowerMeterSeq.iJobReq,
       //                 iPowerMeterHomePos:=#sPowerMeterSeq.iPowerMeterHomePos,
       //                 iPowerMeterWorkPos:=#sPowerMeterSeq.iPowerMeterWorkPos,
       //                 iNC_Stopped:=#sPowerMeterSeq.iNC_Stopped,
       //                 iPLC_DateAndTime:="DB_ReadDateAndTime".sDateAndTime,
       //                 iStepPause:=#sPowerMeterSeq.iStepPause,
       //                 rMinValue:=#sPowerMeterSeq.rMinValue,
       //                 rMaxValue:=#sPowerMeterSeq.rMaxValue,
       //                 iStopOption:=#sPowerMeterSeq.iStopOption,
       //                 rMeasureValue:=#sPowerMeterSeq.rMeasureValue,
       //                 iMeasureDone:=#sPowerMeterSeq.iMeasureDone,
       //                 oPowerMetertoHomeReq=>#sPowerMeterSeq.oPowerMetertoHomeReq,
       //                 oPowerMetertoWorkReq=>#sPowerMeterSeq.oPowerMetertoWorkReq,
       //                 oStopNC_Req=>#sPowerMeterSeq.oStopNC_Req,
       //                 oMsgBadMeasure=>#sPowerMeterSeq.oMsgBadMeasure,
       //                 oStartMeasure=>#sPowerMeterSeq.oStartMeasure,
       //                 oStartArchive=>#sPowerMeterSeq.oStartArchive,
       //                 oRID=>#sPowerMeterSeq.oRID);
   END_REGION

   REGION Powermeter Key / LED Management
       // Disable Powemeter Key[1] if not Jog Mode
       "DB_McpKeyboardSignals".sK1_Powermeter.sKeyDisable := NOT "LBP_ModeGroup".E_JOG OR NOT #tAxis01_X1SafePos OR "DB_GestionWorkingModes".sMCP_KxxKeysDisable;
       "DB_HmiKeyboardSignals".sK1_Powermeter.sKeyDisable := NOT "LBP_ModeGroup".E_JOG OR NOT #tAxis01_X1SafePos;

       // Set/Reset Toggle Powemeter Key[1]
       IF #sPowerMeterSeq.oPowerMetertoWorkReq THEN    // Powermeter to work position
           "DB_McpKeyboardSignals".sK1_Powermeter.sKeySWToggleStatus := TRUE;
           "DB_HmiKeyboardSignals".sK1_Powermeter.sKeySWToggleStatus := TRUE;
       END_IF;
       IF #sPowerMeterSeq.oPowerMetertoHomeReq OR     // Powermeter to home position
           "LBP_Chan1".A_Reset  THEN
           "DB_McpKeyboardSignals".sK1_Powermeter.sKeySWToggleStatus := FALSE;
           "DB_HmiKeyboardSignals".sK1_Powermeter.sKeySWToggleStatus := FALSE;
           END_IF;

       // Powemeter LED[1] Animation
           "DB_McpKeyboardSignals".sK1_Powermeter.sLedSWStatus :=
           ("DB_McpKeyboardSignals".sK1_Powermeter.sKeySWToggleStatus AND #tAxis01_X1SafePos)
           OR ("DB_McpKeyboardSignals".sK1_Powermeter.sKeySWToggleStatus AND "Clock_2Hz");

           "DB_HmiKeyboardSignals".sK1_Powermeter.sLedSWStatus :=
           ("DB_HmiKeyboardSignals".sK1_Powermeter.sKeySWToggleStatus AND #tAxis01_X1SafePos)
           OR ("DB_HmiKeyboardSignals".sK1_Powermeter.sKeySWToggleStatus AND "Clock_2Hz");
   END_REGION

   REGION Powermeter in work position move request
       #sPowerMeterToWorkMoveReq :=
       ("DB_McpKeyboardSignals".sK1_Powermeter.sKeySWToggleStatus AND NOT "MCP1_In".incVar)
       OR ("DB_HmiKeyboardSignals".sK1_Powermeter.sKeySWToggleStatus AND NOT "MCP1_In".incVar)
       AND #tAxis01_X1SafePos;
   END_REGION

   REGION Powermeter in home position move request
       #sPowerMeterToHomeMoveReq :=
       (NOT "DB_McpKeyboardSignals".sK1_Powermeter.sKeySWToggleStatus AND
        NOT "DB_HmiKeyboardSignals".sK1_Powermeter.sKeySWToggleStatus);
   END_REGION

   REGION Powermeter in JOG Mode
       #sPowerMeterJogMode := "LBP_ModeGroup".E_JOG AND "MCP1_Out".LEDincVar;
   END_REGION

   REGION Move/Control Powermeter Cylinder
       #sPowermeterCylinder(iEMinus:="DB_DigitalInputs".sPowerMeterBackCtrl.sSWStatus,
                            iEPlus:="DB_DigitalInputs".sPowerMeterFrontCtrl.sSWStatus,
                            iMinusCmd:=#sPowerMeterToHomeMoveReq,
                            iPlusCmd:=#sPowerMeterToWorkMoveReq,
                            iJOGCmd:=#sPowerMeterJogMode,
                            iMonitorTime:=T#8s,
                            ioQMinus:="DB_DigitalOutputs".sPowerMeterRetract.sSWStatus,
                            ioQPlus:="DB_DigitalOutputs".sPowerMeterAdvance.sSWStatus,
                            oMinusPos=>#sPowermeterInHomePos,
                            oMiddlePos=>#sPowermeterInMiddlePos,
                            oPlusPos=>#sPowermeterInWorkPos,
                            oErrorCode=>#sPowerMeterCylErrorCode);
   END_REGION

   REGION Powermeter Cylinder Positions
       #sPowerMeterHomePos := #sPowermeterCylinder.iEMinus;
       #sPowerMeterWorkPos := #sPowermeterCylinder.iEPlus;
   END_REGION

   REGION Powermeter Cylinder Alarms
       "LBP_AlarmMsgs".UserA[6].A70UUxx[62] := #sPowerMeterCylErrorCode = 1;    // Msg: 700662 "Alarm power meter entry"
       "LBP_AlarmMsgs".UserA[6].A70UUxx[63] := #sPowerMeterCylErrorCode = 2;    // Msg: 700663 "Alarm power meter exit"
   END_REGION

   REGION Monitoring Cylinder in home position
       #sPowerMeterHomePosCtrlTimer(IN:=#sPowerMeterToHomeMoveReq AND NOT #sPowermeterInHomePos,
                                    PT:=#POWERMETER_HOME_POS_CTRL_TIME);

       IF #sPowerMeterHomePosCtrlTimer.Q THEN
           "LBP_AlarmMsgs".ChanA[1].FDD_5C00xx[0] := TRUE;     // Msg: 510000 "Power meter runtimeerror workposition"
       END_IF;

       IF "LBP_Chan1".A_Reset THEN
           "LBP_AlarmMsgs".ChanA[1].FDD_5C00xx[0] := FALSE;    // Msg: 510000 "Power meter runtimeerror workposition"
       END_IF;

       // Read-in disable during movement
       IF #sPowerMeterToHomeMoveReq AND NOT #sPowermeterInHomePos THEN
           "LBP_AlarmMsgs".Chan[1].RID[6] := TRUE;
       END_IF;

       IF #sPowermeterInHomePos OR "LBP_Chan1".A_Reset THEN
           "LBP_AlarmMsgs".Chan[1].RID[6] := FALSE;            
       END_IF;
   END_REGION

   REGION Monitoring Cylinder in work position
       #sPowerMeterWorkPosCtrlTimer(IN := #sPowerMeterToWorkMoveReq AND NOT #sPowermeterInWorkPos,
                                    PT := #POWERMETER_WORK_POS_CTRL_TIME);

       IF #sPowerMeterWorkPosCtrlTimer.Q THEN
           "LBP_AlarmMsgs".ChanA[1].FDD_5C00xx[0] := TRUE;     // Msg: 510000 "Power meter runtimeerror workposition"
       END_IF;

       IF "LBP_Chan1".A_Reset THEN
           "LBP_AlarmMsgs".ChanA[1].FDD_5C00xx[0] := FALSE;    // Msg: 510000 "Power meter runtimeerror workposition"
       END_IF;

       // Read-in disable during movement
       IF #sPowerMeterToWorkMoveReq AND NOT #sPowermeterInWorkPos THEN
           "LBP_AlarmMsgs".Chan[1].RID[7] := TRUE;
       END_IF;

       IF #sPowermeterInWorkPos OR "LBP_Chan1".A_Reset THEN
           "LBP_AlarmMsgs".Chan[1].RID[7] := FALSE;            
       END_IF;
   END_REGION

   REGION Start/Stop measure laser power   
       // M21: Start measure laser power
       IF #sPowerMeterSeq.oStartMeasure THEN
           #sMeasurePowerLaser := TRUE;
       END_IF;

       // M22: Stop measure laser power
       IF NOT #sPowerMeterSeq.oStartMeasure OR "MCP1_In".reset THEN
           #sMeasurePowerLaser := FALSE;
       END_IF;
   END_REGION

   REGION Power value calculation  
       #tLaserMeasureON := #sMeasurePowerLaser OR #sPowerMeterJogMode;

       // Init Powermeter value when restart
       #sRTLaserMeasureON(CLK:=#tLaserMeasureON AND #sPowermeterInWorkPos);
       IF #sRTLaserMeasureON.Q THEN
           #sLaserPowerValue := 0.0;
       END_IF;

       // Power value calculation
       IF #tLaserMeasureON AND #sPowermeterInWorkPos THEN
           #sLaserPowerValue := #sAlpha * "DB_AnalogInputs".sLaserPowerMeter.sSWRealValue +
           (1 - #sAlpha) * #sLaserPowerValue;
           "LBP_NC".A_Setval_anaIn3 := DINT_TO_WORD(REAL_TO_DINT(#sLaserPowerValue * #sWeightFactor));
           "LBP_NC".A_InMask_anaIn3 := TRUE;
       END_IF;
   END_REGION

   REGION Archive 5 last values
       #RT_StartArchive(CLK := #sPowerMeterSeq.oStartArchive);

       IF #RT_StartArchive.Q THEN
           FOR #tIndex := 1 TO 4 DO
               #sArchivePmValues[#tIndex] := #sArchivePmValues[#tIndex - 1];
           END_FOR;
           #sArchivePmValues[0] := #sLaserPowerValue;
       END_IF;
   END_REGION

   REGION Date et Time reading
       #tRetVal := RD_SYS_T(OUT => #sDateAndTime);
   END_REGION

   REGION Measurement archiving
       IF "LBP_Chan1".MDyn[39] THEN
           #tActualMeasure := "DB_PowermeterMeasures".ActualMeasure + 1;
           IF #tActualMeasure >= "DB_PowermeterMeasures".NbMeasure THEN
               #tActualMeasure := 0;
               "DB_PowermeterMeasures".Table_full := TRUE;  // WFA Bit jamais remis à 0
           END_IF;

           "DB_PowermeterMeasures".Measures[#tActualMeasure].Day_meas := DTL_TO_DATE(#sDateAndTime);
           "DB_PowermeterMeasures".Measures[#tActualMeasure].Time_day := DTL_TO_TOD(#sDateAndTime);

           #sActualMeasPower := "LBP_Chan1".H1;

           "DB_PowermeterMeasures".ActualTotalMeas :=
           #sActualMeasPower
           - "DB_PowermeterMeasures".Measures[#tActualMeasure].ValuePower
           + "DB_PowermeterMeasures".ActualTotalMeas;

           "DB_PowermeterMeasures".Measures[#tActualMeasure].ValuePower := #sActualMeasPower;

           REGION Average and Standard Deviation Calculation
               IF "DB_PowermeterMeasures".Table_full THEN
                   #tActualMeasure := 100;
               ELSIF #tActualMeasure < 0 THEN
                   #tActualMeasure := 1;
               END_IF;

               #tAverageValue := "DB_PowermeterMeasures".ActualTotalMeas / #tActualMeasure;

               #tTempReal := ((#tAverageValue * -2.0 * "DB_PowermeterMeasures".ActualTotalMeas) / #tActualMeasure) + #tAverageValue;

               #tStandardDeviation := SQRT(("DB_PowermeterMeasures".ActualMeasure * "DB_PowermeterMeasures".ActualMeasure / #tActualMeasure) + #tTempReal);
           END_REGION

           REGION Compute CM  (" Tol+" - " Tol-" ) / (6 Sigma) process capability index
               IF #tStandardDeviation * 6.0 > 0.0001 THEN
                   #tTempReal := #tStandardDeviation;
               ELSE
                   #tTempReal := 1.0;
               END_IF;

               "DB_PowermeterMeasures".Measures[#tActualMeasure].ValueCM :=
               (#sTolMax - #sTolMin) / #tTempReal;

               "DB_PowermeterMeasures".ActualMeasure := #tActualMeasure;
           END_REGION
       END_IF;
   END_REGION

   REGION Reset Measures
       IF #sResetMeasures THEN
           FOR #tIndex := 0 TO "DB_PowermeterMeasures".NbMeasure - 1 DO
               "DB_PowermeterMeasures".Measures[#tIndex].Job_meas := -1;
               "DB_PowermeterMeasures".Measures[#tIndex].ValuePower := 0.0;
               "DB_PowermeterMeasures".Measures[#tIndex].ValueCM := 0.0;
           END_FOR;
       END_IF;
   END_REGION
END_FUNCTION_BLOCK

FUNCTION_BLOCK "FB_PowerMeterSeq"   // FB92, SCL
{ S7_Optimized_Access := 'TRUE' }
// stored: AutoNumber false, MemoryReserve 100, SetENOAutomatically false
   VAR_INPUT
      iStartSeqCond : Bool;   // Start Sequence Conditions
      iJobReq : Bool;   // Job Request - From Main
      iPowerMeterHomePos : Bool;
      iPowerMeterWorkPos : Bool;
      iNC_Stopped : Bool;
      iPLC_DateAndTime : DTL;
      iStepPause : Bool;
      rMinValue : Real;
      rMaxValue : Real;
      iStopOption : Bool;
      rMeasureValue : Real;
      iMeasureDone : Bool;
   END_VAR
   VAR_OUTPUT
      oPowerMetertoHomeReq { ExternalAccessible := 'False'; ExternalVisible := 'False'; ExternalWritable := 'False'} : Bool;   // Shuttle Start Order - To FB_LoaderAxis
      oPowerMetertoWorkReq { ExternalAccessible := 'False'; ExternalVisible := 'False'; ExternalWritable := 'False'} : Bool;   // Shuttle Position Setpoint - To FB_LoaderAxis
      oStopNC_Req : Bool;
      oMsgBadMeasure : Bool;
      oStartMeasure : Bool;
      oStartArchive : Bool;
      oRID : Bool;
   END_VAR
   VAR
      sCurrent_Step_NB : Int;   // Active Step Number
      sCheck_Step_Condition : Bool;
      sOneStepForward : Bool;
      sRTOneStepForward : R_TRIG;
      sOneStepMode { S7_SetPoint := 'True'} : Bool;
      sStepForward : Bool;
      sInterface : "UDT_SequenceInterface";
      sPowerMetertoHomeReq { ExternalAccessible := 'False'; ExternalVisible := 'False'; ExternalWritable := 'False'} : Bool;
      sPowerMetertoWorkReq { ExternalAccessible := 'False'; ExternalVisible := 'False'; ExternalWritable := 'False'} : Bool;
      sStopNC_Req : Bool;
      sMsgBadMeasure : Bool;
      sStartMeasure : Bool;
      sStartArchive : Bool;
      sMeasureOK : Bool;
      sMeasureNOK : Bool;
      sRID : Bool;
      sHistory : Struct
         Activation : Bool;
         Steps : Array[0..99] of Int;
         Date_Time : Array[0..99] of DTL;
      END_STRUCT;
      StepText : "FB_GetTextErrorCode";
   END_VAR
   VAR_TEMP
      tIndex : Int;   // Index
   END_VAR
   VAR CONSTANT
      S00_INIT : Int := 0;
      S10_SET_RID : Int := 10;
      S20_POWERMETER_TO_WORK_POS : Int := 20;
      S30_START_MEASURE : Int := 30;
      S40_POWERMETER_TO_HOME_POS : Int := 40;
      S50_CHECK_MEASURE : Int := 50;
      S60_RESET_RID : Int := 60;
      S70_SPARE : Int := 70;
      S80_ARCHIVE_MEASURE : Int := 80;
      S160_RESET_RID : Int := 160;
      S170_STOP_CYCLE : Int := 170;
      S180_ARCHIVE_MEASURE : Int := 180;
      S295_JOB_DONE : Int := 295;
   END_VAR
   // StepText.sCode_error[0].ErrorCode := 0;
   // StepText.sCode_error[1].ErrorCode := 10;
   // StepText.sCode_error[2].ErrorCode := 20;
   // StepText.sCode_error[3].ErrorCode := 30;
   // StepText.sCode_error[4].ErrorCode := 40;
   // StepText.sCode_error[5].ErrorCode := 50;
   // StepText.sCode_error[6].ErrorCode := 60;
   // StepText.sCode_error[7].ErrorCode := 70;
   // StepText.sCode_error[8].ErrorCode := 80;
   // StepText.sCode_error[9].ErrorCode := 90;
   // StepText.sCode_error[10].ErrorCode := 95;
BEGIN
   REGION Description header 
       //==================================================================================
       // POSALUX Swiss SA / (C) Copyright 2026
       //----------------------------------------------------------------------------------
       // Title: FB_PowerMeterSeq
       // Comment/Function: 
       // Author: Fabien WALDT
       // Engineering: TIA Portal v20
       //----------------------------------------------------------------------------------
       // Change log table:
       // Version  | Date     | Expert in charge | Changes applied
       // ---------|----------|------------------|-----------------------------------------
       // 00.00.01 | 20260513 | WFA              | First released version
       // =================================================================================
   END_REGION

   REGION Define condition to start
       IF #iStartSeqCond THEN
           #sInterface.SequenceReleased := TRUE;
       ELSE
           // Standard sequencer controls
           #sInterface.SequenceReleased := FALSE;
           #sCurrent_Step_NB := #S00_INIT;
           #sInterface.SequenceRun := FALSE;
           #sInterface.JobDone := FALSE;
           #sCheck_Step_Condition := FALSE;

           // Dedicated sequencer controls
           #sPowerMetertoHomeReq := FALSE;
           #sPowerMetertoWorkReq := FALSE;
           #sStopNC_Req := FALSE;
           #sStartMeasure := FALSE;
           #sStartArchive := FALSE;
           #sMeasureOK := FALSE;
           #sMeasureNOK := FALSE;
           #sRID := FALSE;

           // Add specifics controls 
       END_IF;

       // Reset interface error
       IF #sInterface.Reset THEN
           #sInterface.Error := FALSE;
       END_IF;

       // One step forward
       #sRTOneStepForward.CLK := #sOneStepForward;
       #sRTOneStepForward();
       #sStepForward := (NOT #sOneStepMode OR (#sOneStepMode AND #sRTOneStepForward.Q)) AND NOT #iStepPause;
       #sOneStepForward := FALSE;

       // Action only true in dedicated steps
       #sStopNC_Req := FALSE;
       #sStartMeasure := FALSE;
   END_REGION

   REGION Sequence Function
       CASE #sCurrent_Step_NB OF
           #S00_INIT:
               REGION S00 INIT
                   #sCheck_Step_Condition := TRUE;
                   #sMsgBadMeasure := FALSE;
               END_REGION
           #S10_SET_RID:
               REGION S10_SET_RID
                   #sRID := TRUE;
                   #sCheck_Step_Condition := TRUE;
               END_REGION
           #S20_POWERMETER_TO_WORK_POS:
               REGION S20_POWERMETER_TO_WORK_POS
                   #sPowerMetertoHomeReq := FALSE;
                   #sPowerMetertoWorkReq := TRUE;
                   #sCheck_Step_Condition := TRUE;
               END_REGION
           #S30_START_MEASURE:
               REGION S30_START_MEASURE
                   #sStartMeasure := TRUE;
                   #sCheck_Step_Condition := TRUE;
               END_REGION
           #S40_POWERMETER_TO_HOME_POS:
               REGION S40_POWERMETER_TO_HOME_POS
                   #sPowerMetertoHomeReq := TRUE;
                   #sPowerMetertoWorkReq := FALSE;
                   #sCheck_Step_Condition := TRUE;
               END_REGION
           #S50_CHECK_MEASURE:
               REGION S50_WAIT_OPERATOR_RESTART
                   IF #rMeasureValue <= #rMaxValue AND #rMeasureValue >= #rMinValue THEN
                       #sMeasureOK := TRUE;
                       #sMeasureNOK := FALSE;
                   ELSE
                       #sMeasureOK := FALSE;
                       #sMeasureNOK := TRUE;
                   END_IF;
                   #sCheck_Step_Condition := TRUE;
               END_REGION
           #S60_RESET_RID:
               REGION S60_RESET_RID
                   #sRID := FALSE;
                   #sCheck_Step_Condition := TRUE;
               END_REGION
           #S70_SPARE:
               REGION S70_SPARE
                   #sCheck_Step_Condition := TRUE;
               END_REGION
           #S80_ARCHIVE_MEASURE:
               REGION S80_ARCHIVE_MEASURE
                   #sStartArchive := TRUE;
                   #sCheck_Step_Condition := TRUE;
               END_REGION

           #S160_RESET_RID:
               REGION S160_RESET_RID
                   #sRID := FALSE;
                   #sCheck_Step_Condition := TRUE;
               END_REGION
           #S170_STOP_CYCLE:
               REGION S170_STOP_CYCLE
                   #sStopNC_Req := TRUE;
                   #sCheck_Step_Condition := TRUE;
               END_REGION
           #S180_ARCHIVE_MEASURE:
               REGION S180_ARCHIVE_MEASURE
                   #sStartArchive := TRUE;
                   #sCheck_Step_Condition := TRUE;
               END_REGION

           #S295_JOB_DONE:
               REGION S295_JOB_DONE
                   #sInterface.JobDone := TRUE;
                   #sCheck_Step_Condition := TRUE;
               END_REGION
           ELSE:
               #sInterface.Error := TRUE;
       END_CASE;
   END_REGION

   REGION Sequence Next Step Condition
       IF #sCheck_Step_Condition THEN
           CASE #sCurrent_Step_NB OF
               #S00_INIT:
                   REGION S00 INIT
                       IF #sInterface.SequenceReleased AND #iJobReq THEN
                           #sCurrent_Step_NB := #S10_SET_RID;
                           #sInterface.SequenceRun := TRUE;
                           #sCheck_Step_Condition := FALSE;
                       ELSE
                           #sInterface.SequenceRun := FALSE;
                       END_IF;
                   END_REGION
               #S10_SET_RID:
                   REGION S10_SET_RID
                       IF #sInterface.SequenceReleased AND #sStepForward THEN
                           #sCurrent_Step_NB := #S20_POWERMETER_TO_WORK_POS;
                           #sCheck_Step_Condition := FALSE;
                       END_IF;
                   END_REGION
               #S20_POWERMETER_TO_WORK_POS:
                   REGION S20_POWERMETER_TO_WORK_POS
                       IF #sInterface.SequenceReleased AND #sStepForward AND #iPowerMeterWorkPos THEN
                           #sCurrent_Step_NB := #S30_START_MEASURE;
                           #sCheck_Step_Condition := FALSE;
                       END_IF;
                   END_REGION
               #S30_START_MEASURE:
                   REGION S30_START_MEASURE
                       IF #sInterface.SequenceReleased AND #sStepForward AND #iMeasureDone THEN
                           #sCurrent_Step_NB := #S40_POWERMETER_TO_HOME_POS;
                           #sCheck_Step_Condition := FALSE;
                       END_IF;
                   END_REGION
               #S40_POWERMETER_TO_HOME_POS:
                   REGION S40_POWERMETER_TO_HOME_POS
                       IF #sInterface.SequenceReleased AND #sStepForward AND #iPowerMeterHomePos THEN
                           #sCurrent_Step_NB := #S50_CHECK_MEASURE;
                           #sCheck_Step_Condition := FALSE;
                       END_IF;
                   END_REGION
                   #S50_CHECK_MEASURE:
                       REGION S50_CHECK_MEASURE
                           IF #sInterface.SequenceReleased AND #sStepForward AND (#sMeasureOK OR (#sMeasureNOK AND NOT #iStopOption)) THEN
                               #sCurrent_Step_NB := #S60_RESET_RID;
                               #sCheck_Step_Condition := FALSE;
                           ELSIF #sInterface.SequenceReleased AND #sStepForward AND (#sMeasureNOK AND #iStopOption) THEN
                               #sCurrent_Step_NB := #S160_RESET_RID;
                               #sCheck_Step_Condition := FALSE;
                           END_IF;
                       END_REGION
                   #S60_RESET_RID:
                       REGION S60_RESET_RID
                           IF #sInterface.SequenceReleased AND #sStepForward AND NOT #sRID THEN
                               #sCurrent_Step_NB := #S70_SPARE;
                               #sCheck_Step_Condition := FALSE;
                           END_IF;
                       END_REGION
                   #S70_SPARE:
                       REGION S70_SPARE
                           IF #sInterface.SequenceReleased AND #sStepForward AND "AlwaysTRUE" THEN
                               #sCurrent_Step_NB := #S80_ARCHIVE_MEASURE;
                               #sCheck_Step_Condition := FALSE;
                           END_IF;
                       END_REGION
                   #S80_ARCHIVE_MEASURE:
                       REGION S80_ARCHIVE_MEASURE
                           IF #sInterface.SequenceReleased AND #sStepForward AND "AlwaysTRUE" THEN
                               #sCurrent_Step_NB := #S295_JOB_DONE;
                               #sCheck_Step_Condition := FALSE;
                           END_IF;
                       END_REGION

                   #S160_RESET_RID:
                       REGION S160_RESET_RID
                           IF #sInterface.SequenceReleased AND #sStepForward AND NOT #sRID THEN
                               #sCurrent_Step_NB := #S170_STOP_CYCLE;
                               #sCheck_Step_Condition := FALSE;
                           END_IF;
                       END_REGION
                   #S170_STOP_CYCLE:
                       REGION S170_STOP_CYCLE
                           IF #sInterface.SequenceReleased AND #sStepForward AND #iNC_Stopped THEN
                               #sCurrent_Step_NB := #S180_ARCHIVE_MEASURE;
                               #sCheck_Step_Condition := FALSE;
                           END_IF;
                       END_REGION
                   #S180_ARCHIVE_MEASURE:
                       REGION S180_ARCHIVE_MEASURE
                           IF #sInterface.SequenceReleased AND #sStepForward AND "AlwaysTRUE" THEN
                               #sCurrent_Step_NB := #S295_JOB_DONE;
                               #sCheck_Step_Condition := FALSE;
                           END_IF;
                       END_REGION

                       #S295_JOB_DONE:
                           REGION S295_JOB_DONE
                               IF NOT #iJobReq THEN
                                   #sCurrent_Step_NB := #S00_INIT;
                                   #sCheck_Step_Condition := FALSE;
                                   #sInterface.JobDone := FALSE;
                               END_IF;
                           END_REGION
               ELSE
                   #sInterface.Error := TRUE;
           END_CASE;
       END_IF;
   END_REGION

   REGION Outputs Update
       #oPowerMetertoHomeReq := #sPowerMetertoHomeReq;
       #oPowerMetertoWorkReq := #sPowerMetertoWorkReq;
       #oStopNC_Req := #sStopNC_Req;
       #oMsgBadMeasure := #sMsgBadMeasure;
       #oStartMeasure := #sStartMeasure;
       #oStartArchive := #sStartArchive;
       #oRID := #sRID;
   END_REGION

   REGION Steps - Date and Time History
       IF #sHistory.Activation THEN
           IF #sHistory.Steps[0] <> #sCurrent_Step_NB THEN
               FOR #tIndex := 98 TO 0 BY -1 DO
                   #sHistory.Steps[#tIndex + 1] := #sHistory.Steps[#tIndex];
                   #sHistory.Date_Time[#tIndex + 1] := #sHistory.Date_Time[#tIndex];
               END_FOR;
               #sHistory.Steps[0] := #sCurrent_Step_NB;
               #sHistory.Date_Time[0] := #iPLC_DateAndTime;
           END_IF;
       END_IF;
   END_REGION

   REGION Steps Text
       #StepText(iErrorCode := #sCurrent_Step_NB,
                 oErrorText => #StepText.oErrorText);
   END_REGION
END_FUNCTION_BLOCK

FUNCTION_BLOCK "FB_Pressures"   // FB440, SCL
{ S7_Optimized_Access := 'TRUE' }
// stored: AutoNumber false, IsIECCheckEnabled true, MemoryReserve 100, SetENOAutomatically false
   VAR
      sTimeOutAirDryer : TON_TIME;
      sTimerMachineInDelay : TON_TIME;
      sTimeMachineReadyDelay { S7_SetPoint := 'True'} : TON_TIME;
      sAirInletPressureCtrl { S7_SetPoint := 'True'} : "FB_AnalogInputThreshold";
      sOverpressureScaleZ_Ctrl { S7_SetPoint := 'True'} : "FB_AnalogInputThreshold";
      sOverpressureOpticalPathCtrl { S7_SetPoint := 'True'} : "FB_AnalogInputThreshold";
      sOverpressureLaserHeadCtrl { S7_SetPoint := 'True'} : "FB_AnalogInputThreshold";
      sOverpressureAxisX_Y_Ctrl { S7_SetPoint := 'True'} : "FB_AnalogInputThreshold";
   END_VAR
   VAR CONSTANT
      TIME_OUT_DRYER : Time := T#15S;   // Output short pulse blinking
      TIME_MACHINE_IN_DELAY : Time := T#2S;   // Output short pulse blinking
      OVER_PRESSURE_VALVE_DELAY : Time := T#1S;
      TIME_WAIT_PRESSURE : Time := T#5s;
   END_VAR
BEGIN
   REGION Description header 
       //==================================================================================
       // POSALUX Swiss SA / (C) Copyright 2024
       //----------------------------------------------------------------------------------
       // Title: Management of the pressures of the machine
       // Comment/Function: 
       //
       // Author: Gowsigan SRITHARAN
       // Engineering: TIA Portal v19
       // 
       //----------------------------------------------------------------------------------
       // Change log table:
       // Version  | Date     | Expert in charge | Changes applied
       // ---------|----------|------------------|------------------------------------
       // 00.00.01 | 20250516 | GSR              | First released version
       // ==================================================================================
   END_REGION

   //==================================================================================
   ///////////////////////////////// TECHNICAL TOWER //////////////////////////////////
   // =================================================================================
   REGION Dryer 
       #sTimeOutAirDryer(IN := "DB_PowerOn".sMachineReadySoft AND NOT "DB_DigitalInputs".sAirDryerOK.sSWStatus,
                         PT := #TIME_OUT_DRYER,
                         Q => "LBP_AlarmMsgs".UserA[4].A70UUxx[9]);
   END_REGION

   REGION Air Inlet Pressure
       #sAirInletPressureCtrl(iActualValue:= "DB_AnalogInputs".sInletAirPressure.sSWRealValue,
                              iStartDelay:= "DB_PowerOn".sTimeMachineReadyDelay.Q,
                              ioAlarmMin:= "LBP_AlarmMsgs".UserA[06].A70UUxx[40],
                              ioWarningMin:= "LBP_AlarmMsgs".UserA[07].A70UUxx[40],
                              ioWarningMax:= "LBP_AlarmMsgs".UserA[07].A70UUxx[41],
                              ioAlarmMax:= "LBP_AlarmMsgs".UserA[06].A70UUxx[41],
                              oDataAction=> "DB_AnalogInputAction".Inlet_Air_Pressure,
                              iDataPLC := "DB_AnalogInputDataPLC".Inlet_Air_Pressure,
                              iDataHMI:= "DB_AnalogInputDataHMI".Inlet_Air_Pressure);
   END_REGION

   REGION Output pressure general air
       "DB_DigitalOutputs".sGeneralAirValve.sSWStatus := "DB_PowerOn".sMachineReadySoft;

   END_REGION

   REGION Alarm air pressure
      // pneumatic branching module
       IF "DB_PowerOn".sTimeMachineReadyDelay.Q AND NOT "DB_DigitalInputs".sAirPressureCtrl.sSWStatus THEN
          "LBP_AlarmMsgs".UserA[00].A70UUxx[05] := TRUE;
      END_IF;
   END_REGION

   //==================================================================================
   ///////////////////////////////////// MACHINE //////////////////////////////////////
   //==================================================================================
   REGION Overpressure Scale Z
       #sOverpressureScaleZ_Ctrl(iActualValue:= "DB_AnalogInputs".sZLAxisOverpressure.sSWRealValue,
                                 iStartDelay:= "DB_PowerOn".sTimeMachineReadyDelay.Q,
                                 ioAlarmMin:= "LBP_AlarmMsgs".UserA[06].A70UUxx[42],
                                 ioWarningMin:= "LBP_AlarmMsgs".UserA[07].A70UUxx[42],
                                 ioWarningMax:= "LBP_AlarmMsgs".UserA[07].A70UUxx[43],
                                 ioAlarmMax:= "LBP_AlarmMsgs".UserA[06].A70UUxx[43],
                                 oDataAction=> "DB_AnalogInputAction".ZL_Axis_Overpressure,
                                 iDataPLC := "DB_AnalogInputDataPLC".ZL_Axis_Overpressure,
                                 iDataHMI:= "DB_AnalogInputDataHMI".ZL_Axis_Overpressure);
   END_REGION

   REGION Overpressure Optical path
       #sOverpressureOpticalPathCtrl(iActualValue := "DB_AnalogInputs".sOpticalPathOverpressure.sSWRealValue,
                                     iStartDelay := "DB_PowerOn".sTimeMachineReadyDelay.Q,
                                     ioAlarmMin := "LBP_AlarmMsgs".UserA[06].A70UUxx[44],
                                     ioWarningMin := "LBP_AlarmMsgs".UserA[07].A70UUxx[44],
                                     ioWarningMax := "LBP_AlarmMsgs".UserA[07].A70UUxx[45],
                                     ioAlarmMax := "LBP_AlarmMsgs".UserA[06].A70UUxx[45],
                                     oDataAction=> "DB_AnalogInputAction".Optical_Path_Overpressure,
                                     iDataPLC := "DB_AnalogInputDataPLC".Optical_Path_Overpressure,
                                     iDataHMI := "DB_AnalogInputDataHMI".Optical_Path_Overpressure);
   END_REGION

   REGION Overpressure Laser Head
       #sOverpressureLaserHeadCtrl(iActualValue := "DB_AnalogInputs".sLaserHeadOverpressure.sSWRealValue,
                                   iStartDelay := "DB_PowerOn".sTimeMachineReadyDelay.Q,
                                   ioAlarmMin := "LBP_AlarmMsgs".UserA[06].A70UUxx[46],
                                   ioWarningMin := "LBP_AlarmMsgs".UserA[07].A70UUxx[46],
                                   ioWarningMax := "LBP_AlarmMsgs".UserA[07].A70UUxx[47],
                                   ioAlarmMax := "LBP_AlarmMsgs".UserA[06].A70UUxx[47],
                                   oDataAction=> "DB_AnalogInputAction".Laser_Head_Overpressure,
                                   iDataPLC := "DB_AnalogInputDataPLC".Laser_Head_Overpressure,
                                   iDataHMI := "DB_AnalogInputDataHMI".Laser_Head_Overpressure);
   END_REGION

   REGION Overpressure Axis X and Y
       #sOverpressureAxisX_Y_Ctrl(iActualValue := "DB_AnalogInputs".sXYAxisOverpressure.sSWRealValue,
                                  iStartDelay := "DB_PowerOn".sTimeMachineReadyDelay.Q,
                                  ioAlarmMin := "LBP_AlarmMsgs".UserA[06].A70UUxx[48],
                                  ioWarningMin := "LBP_AlarmMsgs".UserA[07].A70UUxx[48],
                                  ioWarningMax := "LBP_AlarmMsgs".UserA[07].A70UUxx[49],
                                  ioAlarmMax := "LBP_AlarmMsgs".UserA[06].A70UUxx[49],
                                  oDataAction=> "DB_AnalogInputAction".XY_Axis_Overpressure,
                                  iDataPLC := "DB_AnalogInputDataPLC".XY_Axis_Overpressure,
                                  iDataHMI := "DB_AnalogInputDataHMI".XY_Axis_Overpressure);
   END_REGION

   REGION Brake Pressure Ctrl 
       // Reset Channel Feed Disable
       IF "DB_McpKeyboardSignals".sAlarmReset.sKeySWStatus THEN
           "LBP_AlarmMsgs".Chan[1].FDD[9] := FALSE;
       END_IF;

       // X Axis
       IF "DB_PowerOn".sMachinePower
           AND ("LBP_Axis01_X".E_TReqMinus OR "LBP_Axis01_X".E_TReqPlus)
           AND NOT "DB_DigitalInputs".sX_AxisBrakePressCtrl.sSWStatus THEN
           "LBP_AlarmMsgs".UserA[00].A70UUxx[06] := TRUE;
           "LBP_AlarmMsgs".Chan[1].FDD[9] := TRUE;
       END_IF;

       // Y Axis
       IF "DB_PowerOn".sMachinePower
           AND ("LBP_Axis02_Y".E_TReqMinus OR "LBP_Axis02_Y".E_TReqPlus)
           AND NOT "DB_DigitalInputs".sY_AxisBrakePressCtrl.sSWStatus THEN
           "LBP_AlarmMsgs".UserA[00].A70UUxx[07] := TRUE;
           "LBP_AlarmMsgs".Chan[1].FDD[9] := TRUE;
       END_IF;

       // B Axis
       IF "DB_PowerOn".sMachinePower
           AND ("LBP_Axis04_B".E_TReqMinus OR "LBP_Axis04_B".E_TReqPlus)
           AND NOT "DB_DigitalInputs".sB_Axis_BrakeReleasedCtrl.sSWStatus THEN
           "LBP_AlarmMsgs".UserA[00].A70UUxx[08] := TRUE;
           "LBP_AlarmMsgs".Chan[1].FDD[9] := TRUE;
       END_IF;
   END_REGION
END_FUNCTION_BLOCK

FUNCTION_BLOCK "FB_Vacuums"   // FB441, SCL
{ S7_Optimized_Access := 'TRUE' }
// stored: AutoNumber false, MemoryReserve 100, SetENOAutomatically false
   VAR
      sOutVacuum1On : Bool;
      sControlVacuum1 { S7_SetPoint := 'True'} : "FB_AnalogInputThreshold";
      sCtrlPressureVacuum1 { S7_SetPoint := 'True'} : "FB_AnalogInputThreshold";
      sAspirationLeft { S7_SetPoint := 'True'} : "FB_AnalogInputThreshold";
      sAspirationRight { S7_SetPoint := 'True'} : "FB_AnalogInputThreshold";
      sRT_AspirationKeys { S7_SetPoint := 'True'} : R_TRIG;
      sFT_AspirationKeys { S7_SetPoint := 'True'} : F_TRIG;
      sAspirationKeys { S7_SetPoint := 'True'} : Bool;
   END_VAR
BEGIN
   REGION Description header 
       //==================================================================================
       // POSALUX Swiss SA / (C) Copyright 2024
       //----------------------------------------------------------------------------------
       // Title: Vacuums management
       // Comment/Function: This function manages the machine's suction system, controlling
       //                   six suction circuits.
       // Author: Gowsigan SRITHARAN
       // Engineering: TIA Portal v17
       //----------------------------------------------------------------------------------
       // Change log table:
       // Version  | Date     | Expert in charge | Changes applied
       // ---------|----------|------------------|------------------------------------
       // 00.00.01 | 20241120 | GSR              | First released version
       // ---------|----------|------------------|------------------------------------
       // 00.00.02 | 20250327 | WFA              | Management of only one vacuum
       // ==================================================================================
   END_REGION

   REGION Elbaron vacuum
       // Deactivation of the MCP button (MCP Keyboard 9) in Auto mode
       "DB_McpKeyboardSignals".sK9_Aspiration.sKeyDisable := "LBP_ModeGroup".E_AUTO OR "DB_GestionWorkingModes".sMCP_KxxKeysDisable;
       "DB_HmiKeyboardSignals".sK9_Aspiration.sKeyDisable := "LBP_ModeGroup".E_AUTO;

       #sRT_AspirationKeys(CLK := "DB_McpKeyboardSignals".sK9_Aspiration.sKeySWTogglePositiveFront
                           OR "DB_HmiKeyboardSignals".sK9_Aspiration.sKeySWTogglePositiveFront);

       #sFT_AspirationKeys(CLK := "DB_McpKeyboardSignals".sK9_Aspiration.sKeySWToggleNegativeFront
                           OR "DB_HmiKeyboardSignals".sK9_Aspiration.sKeySWToggleNegativeFront);

       IF #sRT_AspirationKeys.Q THEN
           #sAspirationKeys := TRUE;
       ELSIF #sFT_AspirationKeys.Q THEN
           #sAspirationKeys := FALSE;
       END_IF;

       // Activation of the Elbaron output
       "DB_DigitalOutputs".sElbaronPowerON.sSWStatus :=
       "DB_PowerOn".sMachineReadySoft
       AND NOT "DB_Machineshutdown_UPS".sShutDownAspiration
       AND ((("LBP_Chan1".E_ProgRunning
       OR "LBP_Chan1".E_ProgWait
       OR "LBP_Chan1".E_ProgStop
       OR "LBP_Chan2".E_ProgRunning
       OR "LBP_Chan2".E_ProgWait
       OR "LBP_Chan2".E_ProgStop)
       AND "LBP_ModeGroup".E_AUTO)
       OR #sAspirationKeys);

       // Keys Elbaron Aspiration
       "DB_McpKeyboardSignals".sK9_Aspiration.sKeySWToggleStatus := "DB_DigitalOutputs".sElbaronPowerON.sSWStatus;
       "DB_HmiKeyboardSignals".sK9_Aspiration.sKeySWToggleStatus := "DB_DigitalOutputs".sElbaronPowerON.sSWStatus;

       // LED Elbaron Aspiration
       "DB_McpKeyboardSignals".sK9_Aspiration.sLedSWStatus := "DB_DigitalOutputs".sElbaronPowerON.sSWStatus;
       "DB_HmiKeyboardSignals".sK9_Aspiration.sLedSWStatus := "DB_DigitalOutputs".sElbaronPowerON.sSWStatus;
   END_REGION

   REGION Aspirations control
       #sAspirationLeft(iActualValue := "DB_AnalogInputs".sLeftAspiration.sSWRealValue,
                        iStartDelay := "DB_DigitalOutputs".sElbaronPowerON.sSWStatus,
                        ioAlarmMin := "LBP_AlarmMsgs".UserA[06].A70UUxx[56],
                        ioWarningMin := "LBP_AlarmMsgs".UserA[07].A70UUxx[56],
                        ioWarningMax := "LBP_AlarmMsgs".UserA[07].A70UUxx[57],
                        ioAlarmMax := "LBP_AlarmMsgs".UserA[06].A70UUxx[57],
                        oDataAction => "DB_AnalogInputAction".Left_Aspiration,
                        iDataPLC := "DB_AnalogInputDataPLC".Left_Aspiration,
                        iDataHMI := "DB_AnalogInputDataHMI".Left_Aspiration);

       #sAspirationRight(iActualValue := "DB_AnalogInputs".sRightAspiration.sSWRealValue,
                         iStartDelay := "DB_DigitalOutputs".sElbaronPowerON.sSWStatus,
                         ioAlarmMin := "LBP_AlarmMsgs".UserA[06].A70UUxx[58],
                         ioWarningMin := "LBP_AlarmMsgs".UserA[07].A70UUxx[58],
                         ioWarningMax := "LBP_AlarmMsgs".UserA[07].A70UUxx[59],
                         ioAlarmMax := "LBP_AlarmMsgs".UserA[06].A70UUxx[59],
                         oDataAction => "DB_AnalogInputAction".Right_Aspiration,
                         iDataPLC := "DB_AnalogInputDataPLC".Right_Aspiration,
                         iDataHMI := "DB_AnalogInputDataHMI".Right_Aspiration);
   END_REGION
END_FUNCTION_BLOCK

FUNCTION_BLOCK "FB_Cognex"   // FB55, SCL
{ S7_Optimized_Access := 'TRUE' }
// stored: AutoNumber false, MemoryReserve 100, SetENOAutomatically false
   VAR
      sASTriggerReadyMemo : Bool;
      sASTriggerAckMemo : Bool;
      sASAcquiringMemo : Bool;
      sASMissedTrigMemo : Bool;
      sASOfflineResBit1Memo : Bool;
      sASOfflineResBit2Memo : Bool;
      sASOfflineResBit3Memo : Bool;
      sASOnlineMemo : Bool;
      sISInspectingMemo : Bool;
      sISToggleInspectDoneMemo : Bool;
      sISBufferOverrunMemo : Bool;
      sISResultsValidMemo : Bool;
      sISJobLoadingMemo : Bool;
      sISJobLoadCompleteMemo : Bool;
      sISJobLoadFailedMemo : Bool;
      sISSetUserDataACkMemo : Bool;
      sISJobPassMemo : Bool;
      sSEC0AckMemo : Bool;
      sSEC1AckMemo : Bool;
      sSEC2AckMemo : Bool;
      sSEC3AckMemo : Bool;
      sSEC4AckMemo : Bool;
      sSEC5AckMemo : Bool;
      sSEC6AckMemo : Bool;
      sSEC7AckMemo : Bool;
      sACTriggerEnableMemo : Bool;
      sACTriggerMemo : Bool;
      sACClearAcquirComplMemo : Bool;
      sACSetOfflineMemo : Bool;
      sICBufferResultsEnMemo : Bool;
      sICInspectResultsAckMemo : Bool;
      sICSetUserDataMemo : Bool;
      sICExecuteCmdMemo : Bool;
      sCCSetJobIDMemo : Int;
      sSEC0Memo : Bool;
      sSEC1Memo : Bool;
      sSEC2Memo : Bool;
      sSEC3Memo : Bool;
      sSEC4Memo : Bool;
      sSEC5Memo : Bool;
      sSEC6Memo : Bool;
      sSEC7Memo : Bool;
      sCamLightOn : Bool;
      sUserDataWrite : Bool;
      sUserDataWriteEn : Bool;
      sStartCapture : Bool;
      sAfterResultSoft7 : Bool;
      sTrigAckMemory : Bool;
      sMemoM55 : Bool;
      sSetSetup : Bool;
      sResultDataErrorBit : Bool;
      sICBufferResultsEnPositiveFront : Bool;
      sUserResultReadHole : Bool;
      sUserDataErrorBit : Bool;
      sIRActHoleNrResultMemo : Byte;
      sSetJobId : Int;
      sSetJobIdMemo : Int;
      sJCJobIDMemo : Word;
      sIRInspectionIDMemo : Word;
      sIRInspectResultCodeMemo : Word;
      sASAcquiNumMemo : Word;
      sUserDataErrorCode : Int;
      sResultDataErrorCode : Int;
      sNumChannel : Int;
      sCountAcquiNr : Int;
      sCounter : CTUD_INT;
      sUserDataArray : Array[0..7] of DWord;
      sResultDataArray : Array[0..3] of DWord;
   END_VAR
BEGIN
   REGION Acquisition status
       #sASTriggerReadyMemo := "ASTriggerReady";
       #sASTriggerAckMemo := "ASTriggerAck";
       #sASAcquiringMemo := "ASAcquiring";
       #sASMissedTrigMemo := "ASMissedTrig";
       #sASOfflineResBit1Memo := "ASOfflineResBit1";
       #sASOfflineResBit2Memo := "ASOfflineResBit2";
       #sASOfflineResBit3Memo := "ASOfflineResBit3";
       #sASOnlineMemo := "ASOnline";
       #sASAcquiNumMemo := "ASAcquiNum";
   END_REGION

   REGION Inspection status
       #sISInspectingMemo := "ISInspecting";
       #sISToggleInspectDoneMemo := "ISToggleInspectDone";
       #sISBufferOverrunMemo := "ISBufferOverrun";
       #sISResultsValidMemo := "ISResultsValid";
       #sISJobLoadingMemo := "ISJobLoading";
       "LBP_AlarmMsgs".UserA[8].A70UUxx[41] := "ISJobLoading";
       #sISJobLoadCompleteMemo := "ISJobLoadComplete";
       #sISJobLoadFailedMemo := "ISJobLoadFailed";
       #sISSetUserDataACkMemo := "ISSetUserDataACk";
       #sISJobPassMemo := "ISJobPass";
   END_REGION

   REGION Soft event control output MODule
       #sSEC0AckMemo := "SEC0Ack";
       #sSEC1AckMemo := "SEC1Ack";
       #sSEC2AckMemo := "SEC2Ack";
       #sSEC3AckMemo := "SEC3Ack";
       #sSEC4AckMemo := "SEC4Ack";
       #sSEC5AckMemo := "SEC5Ack";
       #sSEC6AckMemo := "SEC6Ack";
       #sSEC7AckMemo := "SEC7Ack";
   END_REGION

   REGION Job control
       #sJCJobIDMemo := "JCJobID";
   END_REGION

   REGION Inspection result
       #sIRInspectionIDMemo := "IRInspectionID";
       #sIRInspectResultCodeMemo := "IRInspectResultCode";

   END_REGION


   REGION Part programme <-> cognex
       IF #sASOnlineMemo THEN
           // RID if missed trig
           "LBP_AlarmMsgs".ChanA[1].FDD_RID_5C01xx[10] := #sICBufferResultsEnMemo AND #sASMissedTrigMemo;

           // Start camera and set buffer valid
           IF "LBP_Chan1".MDyn[52] THEN    // M52 : Enable buffer and restart the counter hole
               #sICBufferResultsEnMemo := TRUE;
               #sACTriggerEnableMemo := TRUE;
               "LBP_AlarmMsgs".Chan[1].RID[0] := TRUE;
               #sSEC5Memo := FALSE;
           END_IF;

           IF #sASTriggerReadyMemo THEN
               "LBP_AlarmMsgs".Chan[1].RID[0] := FALSE;
           END_IF;

           IF "LBP_Chan1".A_Reset THEN
               #sICBufferResultsEnMemo := FALSE;
               #sACTriggerEnableMemo := FALSE;
               "LBP_AlarmMsgs".Chan[1].RID[0] := FALSE;
               #sSEC5Memo := FALSE;
           END_IF;

           // M53 holes param to Cognex and start capture
           IF "LBP_Chan1".MDyn[53] THEN
               #sUserDataWrite := TRUE;
               #sUserDataWriteEn := TRUE;
               "LBP_AlarmMsgs".Chan[1].RID[11] := TRUE;
           END_IF;

           IF "LBP_Chan1".A_Reset THEN
               #sUserDataWrite := FALSE;
               #sUserDataWriteEn := FALSE;
               "LBP_AlarmMsgs".Chan[1].RID[11] := FALSE;
               #sStartCapture := FALSE;
           END_IF;

           // M54 start acquisition
           IF "LBP_Chan1".MDyn[54] THEN
               #sStartCapture := TRUE;
               "LBP_AlarmMsgs".Chan[1].RID[1] := TRUE;
           END_IF;

           #sACClearAcquirComplMemo :="LBP_Chan1".MDyn[54];

           #sCounter.CU := #sStartCapture AND #sASTriggerReadyMemo AND NOT #sCounter.QU;

           IF #sStartCapture AND #sASTriggerReadyMemo AND NOT #sCounter.QU THEN
               #sACTriggerMemo := TRUE;
               #sAfterResultSoft7 := TRUE;
           END_IF;

           IF #sASTriggerAckMemo THEN
               #sACTriggerMemo := FALSE;
               #sTrigAckMemory := TRUE;
           END_IF;

           IF #sTrigAckMemory AND #sASAcquiringMemo THEN
               #sStartCapture := FALSE;
               "LBP_AlarmMsgs".Chan[1].RID[1] := FALSE;
               #sTrigAckMemory := FALSE;
           END_IF;

           #sCounter.R := "LBP_Chan1".A_Reset;

           IF "LBP_Chan1".A_Reset THEN
               "LBP_AlarmMsgs".Chan[1].RID[1] := FALSE;
               #sACTriggerMemo := FALSE;
           END_IF;

           // M55 end measure
           IF "LBP_Chan1".MDyn[55] AND #sICBufferResultsEnMemo THEN
               "LBP_AlarmMsgs".Chan[1].RID[2] := TRUE;
               #sMemoM55 := TRUE;
               #sSEC6Memo := FALSE;
           END_IF;

           IF (#sMemoM55 AND NOT #sCounter.QU) OR "LBP_Chan1".A_Reset THEN
               #sMemoM55 := FALSE;
               #sACTriggerEnableMemo := FALSE;
               #sSEC5Memo := TRUE;
           END_IF;

           IF #sSEC5AckMemo THEN
               #sSEC5Memo := FALSE;
           END_IF;

               // End part programme <-> cognex
               "LBP_AlarmMsgs".UserA[8].A70UUxx[0] := FALSE;
               "LBP_AlarmMsgs".Chan[1].RID[3] := FALSE;

       ELSE
           IF "LBP_Chan1".MDyn[52]
               OR "LBP_Chan1".MDyn[53]
               OR "LBP_Chan1".MDyn[54]
               OR "LBP_Chan1".MDyn[55] THEN
               "LBP_AlarmMsgs".UserA[8].A70UUxx[0] := TRUE;
               "LBP_AlarmMsgs".Chan[1].RID[3] := TRUE;
           END_IF;

           IF "LBP_Chan1".A_Reset THEN
                "LBP_AlarmMsgs".UserA[8].A70UUxx[0] := FALSE;
                "LBP_AlarmMsgs".Chan[1].RID[3] := FALSE;
           END_IF;

       END_IF;
   END_REGION

   REGION Inspection control
       IF #sISSetUserDataACkMemo AND #sICSetUserDataMemo THEN
           #sICSetUserDataMemo := FALSE;
           #sSEC6Memo := FALSE;
       END_IF;

       IF #sSEC6Memo AND #sSEC6AckMemo THEN
           #sSEC6Memo := FALSE;
           "LBP_AlarmMsgs".Chan[1].RID[11] := FALSE;
       END_IF;
   END_REGION



   REGION Acquisition control
       "ACTriggerEnable" := #sACTriggerEnableMemo;
       "ACTrigger" := #sACTriggerMemo;
       "ACClearAcquirCompl" := #sACClearAcquirComplMemo;
       "ACSetOffline" := #sACSetOfflineMemo;
   END_REGION

   REGION Inspection control
       "ICBufferResultsEn" := #sICBufferResultsEnMemo;
       "ICInspectResultsAck" := #sICInspectResultsAckMemo;
       "ICSetUserData" := #sICSetUserDataMemo;
       "ICExecuteCmd" := #sICExecuteCmdMemo;

       IF #sISSetUserDataACkMemo AND #sICSetUserDataMemo THEN
           #sICSetUserDataMemo := FALSE;
           #sSEC6Memo := TRUE;
       END_IF;

       IF #sSEC6AckMemo AND #sSEC6Memo THEN
           #sSEC6Memo := FALSE;
           "LBP_AlarmMsgs".Chan[1].RID[11] := FALSE;
       END_IF;

   END_REGION

   REGION Job control in setup
       IF "LBP_Chan1".MDyn[58] THEN
           #sSetSetup := TRUE;
           "LBP_AlarmMsgs".Chan[1].RID[13] := TRUE;
       ELSE
           #sSetJobId :=  REAL_TO_INT(ROUND("LBP_Chan1".H1));
       END_IF;

       IF "LBP_Chan1".MDyn[59] THEN
           #sSetSetup := FALSE;
           "LBP_AlarmMsgs".Chan[1].RID[13] := TRUE;
       END_IF;

       IF "LBP_Chan1".A_Reset THEN
           #sSetSetup := FALSE;
           "LBP_AlarmMsgs".Chan[1].RID[13] := FALSE;
           #sICExecuteCmdMemo := FALSE;
           #sACSetOfflineMemo := FALSE;
       END_IF;

   END_REGION

   REGION Job control
       IF #sSetSetup THEN
           // Set new job
           #sSetJobIdMemo := #sSetJobId;
           // If actual job in camera is not the new one AND cmd in progress
           IF NOT (#sSetJobIdMemo = #sJCJobIDMemo
               AND NOT "ICExecuteCmd") THEN
               // Set offline to load job
               IF #sASOnlineMemo THEN
                   #sACSetOfflineMemo := TRUE;
               ELSE
                   // Load job
                   IF NOT #sICExecuteCmdMemo THEN
                       #sCCSetJobIDMemo := #sSetJobIdMemo;
                       #sICExecuteCmdMemo := TRUE;
                   ELSE
                       // Wait job is loaded
                       IF #sISJobLoadCompleteMemo THEN
                           // Reset cmd
                           #sICExecuteCmdMemo := FALSE;
                           #sACSetOfflineMemo := FALSE;
                           "LBP_AlarmMsgs".Chan[1].RID[13] := FALSE;
                           // If load failed
                           IF #sISJobLoadFailedMemo THEN
                               #sICExecuteCmdMemo := FALSE;
                               #sACSetOfflineMemo := FALSE;
                           END_IF;
                       END_IF;
                    END_IF;
               END_IF;
           END_IF;
       END_IF;

   END_REGION

   REGION Soft event control
       "SEC0" := #sSEC0Memo;
       "SEC1" := #sSEC1Memo;
       "SEC2" := #sSEC2Memo;
       "SEC3" := #sSEC3Memo;
       "SEC4" := #sSEC4Memo;
       "SEC5" := #sSEC5Memo;
       "SEC6" := #sSEC6Memo;
       "SEC7" := #sSEC7Memo;

       IF "LBP_Chan1".MDyn[55] OR "LBP_Chan1".A_Reset THEN
           #sSEC0Memo := FALSE;
           #sSEC1Memo := FALSE;
           #sSEC2Memo := FALSE;
           #sSEC3Memo := FALSE;
           #sSEC4Memo := FALSE;
           //#SEC5Memo := FALSE;
           #sSEC6Memo := FALSE;
           #sSEC7Memo := FALSE;
       END_IF;
   END_REGION

   REGION User data from NC
       // If part program send M code
       IF #sUserDataWrite THEN
           // Read data from part program
           "LBP_TransferSelData"(Enable:=#sUserDataWrite,
                                 Funct:=B#16#3,
                                 IVAR1:=8,
                                 IVAR2:=-1,
                                 Error=>#sUserDataErrorBit,
                                 ErrCode=>#sUserDataErrorCode,
                                 S7Var:=#sUserDataArray);

           IF NOT #sUserDataErrorBit THEN
               "UserDataToCognex0" := #sUserDataArray[0];
               "UserDataToCognex1" := #sUserDataArray[1];
               "UserDataToCognex2" := #sUserDataArray[2];
               "UserDataToCognex3" := #sUserDataArray[3];
               "UserDataToCognex4" := #sUserDataArray[4];
               "UserDataToCognex5" := #sUserDataArray[5];
               "UserDataToCognex6" := #sUserDataArray[6];
               "UserDataToCognex7" := #sUserDataArray[7];
           END_IF;

           IF #sUserDataWriteEn AND NOT #sUserDataWrite THEN
               #sUserDataWrite := FALSE;
           END_IF;

           IF #sUserDataWriteEn AND NOT #sUserDataErrorBit THEN
               #sICSetUserDataMemo := FALSE;
               #sUserDataWrite := FALSE;
           END_IF;
       END_IF;

   END_REGION

   REGION Result data to NC
       // Check if cognex has something new
       IF #sISResultsValidMemo AND #sICBufferResultsEnMemo AND NOT #sICBufferResultsEnPositiveFront THEN
           #sUserResultReadHole := TRUE;

           IF #sAfterResultSoft7 THEN
               #sAfterResultSoft7 := FALSE;
               #sSEC4Memo := TRUE;
           END_IF;

           // Define which hole
           IF "IRActHoleNrResult" < 10 THEN
               #sIRActHoleNrResultMemo := "IRActHoleNrResult";
           ELSE
               #sIRActHoleNrResultMemo := 1;
           END_IF;

           #sNumChannel := #sIRActHoleNrResultMemo * 16 + 40;

           // Send result to part program
           #sResultDataArray[0] := "ResultDataFromCognex0";
           #sResultDataArray[1] := "ResultDataFromCognex1";
           #sResultDataArray[2] := "ResultDataFromCognex2";
           #sResultDataArray[3] := "ResultDataFromCognex3";

           "LBP_TransferSelData"(Enable := #sUserResultReadHole,
                                 Funct := B#16#4,
                                 IVAR1 := #sNumChannel,
                                 IVAR2 := -1,
                                 Error => #sResultDataErrorBit,
                                 ErrCode => #sUserDataErrorCode,
                                 S7Var := #sResultDataArray);


       END_IF;

       // Acknowledgements
       #sICBufferResultsEnPositiveFront := #sICBufferResultsEnMemo;

       #sCounter.CD := NOT #sResultDataErrorBit AND #sUserResultReadHole;

       IF NOT #sResultDataErrorBit AND #sUserResultReadHole THEN
           #sUserResultReadHole := FALSE;
           #sICInspectResultsAckMemo := TRUE;

       END_IF;

       #sCountAcquiNr := #sCounter.CV;

       IF NOT #sISResultsValidMemo OR "LBP_Chan1".A_Reset THEN
           #sICInspectResultsAckMemo := FALSE;
       END_IF;

       IF #sSEC4AckMemo THEN
           #sSEC4Memo := FALSE;
       END_IF;

       IF "LBP_Chan1".A_Reset THEN
           #sUserResultReadHole := FALSE;
       END_IF;
   END_REGION
END_FUNCTION_BLOCK

FUNCTION_BLOCK "FB_Machineshutdown_UPS"   // FB461, SCL
{ S7_Optimized_Access := 'TRUE' }
// stored: AutoNumber false, MemoryReserve 100, SetENOAutomatically false
   VAR
      sTimeOutShutDown { S7_SetPoint := 'True'} : TON_TIME;
      sTimeOutAlarmUPS { S7_SetPoint := 'True'} : TON_TIME;
      sTimeOutShutDownPC { S7_SetPoint := 'True'} : TON_TIME;
      sShutDownDelayPC { S7_SetPoint := 'True'} : TON_TIME;
      sShutDownAspiration : Bool;
      sShutDownPower : Bool;
      sShutDownPCRequest : Int;
      sShutDownPCResponse : Int;
   END_VAR
   VAR CONSTANT
      TIME_OUT_SHUTDOWN : Time := T#3S;
      TIME_OUT_ALARM_UPS : Time := T#30S;
      TIME_OUT_SHUTDOWN_PC : Time := T#7M;
      DELAY_SHUTDOWN_PC : Time := T#1M;
   END_VAR
BEGIN
   REGION Shutdown Machine
       // Time out button shutdown and ups Alarm
       #sTimeOutAlarmUPS.TON(IN := NOT "DB_DigitalInputs".sUPS_PowerFailure.sSWStatus AND NOT "DB_DigitalInputs".sUPS_CommonAlarm.sSWStatus,
                             PT := #TIME_OUT_ALARM_UPS);
       #sTimeOutShutDown.TON(IN := "DB_McpKeyboardSignals".sShutdownPC.sKeySWStatus,
                             PT := #TIME_OUT_SHUTDOWN);
       #sTimeOutShutDownPC.TON(IN := #sShutDownPCRequest <> 0 AND #sShutDownPCResponse <> 1,
                               PT := #TIME_OUT_SHUTDOWN_PC);
       #sShutDownDelayPC.TON(IN := #sShutDownPCResponse = 1,
                             PT := #DELAY_SHUTDOWN_PC);

       // Send request to Left_PC
       IF #sTimeOutShutDown.Q THEN
           #sShutDownPCRequest := 1;
           "LBP_AlarmMsgs".UserA[4].A70UUxx[42] := NOT "LBP_AlarmMsgs".UserA[4].A70UUxx[41];
       ELSIF #sTimeOutAlarmUPS.Q THEN
           // Power Failure
           #sShutDownPCRequest := 2;
           "LBP_AlarmMsgs".UserA[4].A70UUxx[23] := TRUE;
       END_IF;

       // Management of signal feedback or timeout
       IF #sShutDownDelayPC.Q THEN
           // Machine stop process completed. Turn off the machine using the main switch
           "LBP_AlarmMsgs".UserA[4].A70UUxx[41] := NOT "DB_PowerOn".sMachineReadySoft; // Message pour couper l'alimentation si BT jaune extinction
           "DB_DigitalOutputs".sEPO_UPS.sSWStatus := #sShutDownPCRequest = 2;          // Ouverture du relais EPO si UPS extinction
       ELSIF #sShutDownPCResponse = 1 THEN
           #sShutDownPower := true;
       ELSIF #sShutDownPCResponse = 2 THEN
           // Laser status unknown. Turn it off on left PC THEN wait FOR the machine's shutdown
           "LBP_AlarmMsgs".UserA[4].A70UUxx[22] := TRUE;
       ELSIF #sShutDownPCResponse = 3 THEN
           // The laser is still on. Please turn it off manually
           "LBP_AlarmMsgs".UserA[4].A70UUxx[21] := TRUE;
       ELSIF #sShutDownPCResponse = 4 THEN
           #sShutDownAspiration := TRUE;
       ELSIF #sTimeOutShutDownPC.Q THEN
           // Timeout shutdown. Please turn it off manually
           "LBP_AlarmMsgs".UserA[4].A70UUxx[20] := TRUE;
       END_IF;

       // Shutdown Button LED
       "DB_McpKeyboardSignals".sShutdownPC.sLedSWStatus :=
       ("DB_McpKeyboardSignals".sShutdownPC.sKeySWStatus AND "Clock_5Hz")
       OR (#sShutDownPCRequest <> 0 AND #sShutDownPCResponse <> 1)
       OR #sShutDownPower
       OR "DB_McpKeyboardSignals".sLightTest.sKeySWStatus;
   END_REGION


   REGION UPS Alarms
       IF "DB_MachineOptions".UPSPresent THEN
           IF "DB_DigitalInputs".sUPS_BatteryLow.sSWStatus
               AND NOT "DB_DigitalInputs".sUPS_BatteryOK.sSWStatus THEN
               "LBP_AlarmMsgs".UserA[4].A70UUxx[2] := TRUE;
           END_IF;

           IF NOT "DB_DigitalInputs".sUPS_ByPassActive.sSWStatus THEN
               "LBP_AlarmMsgs".UserA[4].A70UUxx[3] := TRUE;
           END_IF;

           IF NOT "DB_DigitalInputs".sUPS_Fault.sSWStatus
               OR NOT "DB_DigitalInputs".sUPS_CommonAlarm.sSWStatus THEN
               "LBP_AlarmMsgs".UserA[4].A70UUxx[4] := TRUE;
           END_IF;

           IF NOT "DB_DigitalInputs".sUPS_PowerFailure.sSWStatus
               AND NOT "DB_DigitalInputs".sUPS_CommonAlarm.sSWStatus THEN
               "LBP_AlarmMsgs".UserA[4].A70UUxx[5] := TRUE;
           END_IF;

           IF "DB_DigitalInputs".sInverterActive.sSWStatus THEN
               "LBP_AlarmMsgs".UserA[4].A70UUxx[6] := TRUE;
           END_IF;
       END_IF;
   END_REGION
END_FUNCTION_BLOCK

